KUKA KRL program: MyProgram_232().src

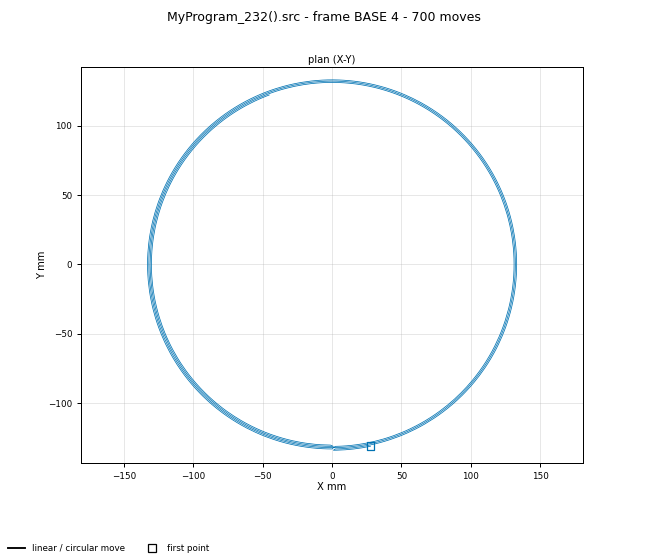
[picture p0: tool path of MyProgram_232().src in frame BASE 4, 700 of 700 moves have a stored position in this frame; points joined in program order, loops and branches not executed]
&ACCESS RVP
&REL 1
&PARAM TEMPLATE = C:\KRC\Roboter\Template\vorgabe
&PARAM EDITMASK = *
DEF MyProgram_232()
; ---- Setting reference (Base) ----
$BASE = BASE_DATA[4]

; --------------------------
; ---- Setting tool (TCP) ----
$TOOL = TOOL_DATA[3]
; --------------------------

$VEL.CP = VEL_APROX_PRINT
Startdeposition()
$VEL.CP = VEL_PRINT
LIN {X 27.6875,Y -131.1265,Z 158,A -80.2981,B 21.5066,C -0.6867,E1 21.5496,E2 528.0093} C_DIS
LIN {X 24.3865,Y -131.7813,Z 158,A -81.7242,B 21.5066,C -0.6861,E1 21.5457,E2 529.435} C_DIS
LIN {X 21.7115,Y -132.2465,Z 158,A -82.8486,B 21.5066,C -0.6869,E1 21.5426,E2 530.5558} C_DIS
LIN {X 18.7326,Y -132.701,Z 158,A -84.1707,B 21.5067,C -0.6845,E1 21.5389,E2 531.883} C_DIS
LIN {X 15.6602,Y -133.0985,Z 158,A -85.5143,B 21.5067,C -0.6828,E1 21.5352,E2 533.2299} C_DIS
LIN {X 12.3449,Y -133.4475,Z 158,A -86.8751,B 21.5067,C -0.685,E1 21.5314,E2 534.5836} C_DIS
LIN {X 9.7078,Y -133.6645,Z 158,A -88.0842,B 21.5068,C -0.681,E1 21.528,E2 535.8031} C_DIS
LIN {X 6.5931,Y -133.8544,Z 158,A -89.4325,B 21.5068,C -0.6798,E1 21.5243,E2 537.1539} C_DIS
LIN {X 3.271,Y -133.9775,Z 158,A -90.7812,B 21.5068,C -0.6827,E1 21.5205,E2 538.4945} C_DIS
LIN {X 0.9335,Y -134.0118,Z 158,A -91.4761,B 21.5063,C -0.6963,E1 21.5187,E2 539.1521} C_DIS
Enddeposition()
LIN {X 0.9335,Y -134.0118,Z 158,A -91.4761,B 21.5063,C -0.6963,E1 21.5187,E2 539.1521} C_DIS
Startdeposition()
$VEL.CP = VEL_PRINT
LIN {X 2.3152,Y -133.0672,Z 158,A -90.1607,B 20.3364,C -0.5545,E1 20.3481,E2 538.1148} C_DIS
LIN {X 6.4619,Y -132.9305,Z 158,A -88.4091,B 20.3364,C -0.5536,E1 20.353,E2 536.3665} C_DIS
LIN {X 10.2986,Y -132.6896,Z 158,A -86.7068,B 20.3364,C -0.5563,E1 20.3578,E2 534.6574} C_DIS
LIN {X 14.1975,Y -132.3277,Z 158,A -85.0987,B 20.3364,C -0.5538,E1 20.3622,E2 533.0578} C_DIS
LIN {X 17.9935,Y -131.867,Z 158,A -83.332,B 20.3363,C -0.56,E1 20.3671,E2 531.2751} C_DIS
LIN {X 21.7924,Y -131.2908,Z 158,A -81.8494,B 20.3364,C -0.5537,E1 20.3712,E2 529.8124} C_DIS
LIN {X 26.2701,Y -130.4688,Z 158,A -79.804,B 20.3364,C -0.559,E1 20.3768,E2 527.7549} C_DIS
LIN {X 29.9306,Y -129.678,Z 158,A -78.1545,B 20.3362,C -0.562,E1 20.3813,E2 526.0995} C_DIS
LIN {X 34.3931,Y -128.5662,Z 158,A -76.2181,B 20.3362,C -0.562,E1 20.3866,E2 524.1667} C_DIS
LIN {X 37.8734,Y -127.5852,Z 158,A -74.6229,B 20.3362,C -0.5654,E1 20.3908,E2 522.5654} C_DIS
LIN {X 41.9126,Y -126.315,Z 158,A -72.8787,B 20.3362,C -0.564,E1 20.3955,E2 520.8291} C_DIS
LIN {X 45.0525,Y -125.2293,Z 158,A -71.5317,B 20.3362,C -0.5621,E1 20.399,E2 519.491} C_DIS
LIN {X 48.0237,Y -124.1204,Z 158,A -70.214,B 20.3362,C -0.5618,E1 20.4024,E2 518.1778} C_DIS
LIN {X 50.4919,Y -123.1393,Z 158,A -68.8394,B 20.3359,C -0.5736,E1 20.406,E2 516.7734} C_DIS
LIN {X 54.0949,Y -121.5973,Z 158,A -67.513,B 20.3363,C -0.5601,E1 20.4093,E2 515.4899} C_DIS
LIN {X 57.1818,Y -120.1764,Z 158,A -65.8004,B 20.3359,C -0.5733,E1 20.4138,E2 513.7447} C_DIS
LIN {X 60.0472,Y -118.771,Z 158,A -64.3224,B 20.3357,C -0.5801,E1 20.4175,E2 512.2522} C_DIS
LIN {X 63.9135,Y -116.7378,Z 158,A -62.5187,B 20.3357,C -0.5798,E1 20.4219,E2 510.4559} C_DIS
LIN {X 66.8745,Y -115.0672,Z 158,A -60.0156,B 20.3343,C -0.6293,E1 20.4283,E2 507.8206} C_DIS
LIN {X 73.3086,Y -111.0787,Z 158,A -57.8118,B 20.3355,C -0.5876,E1 20.4331,E2 505.7453} C_DIS
LIN {X 76.8539,Y -108.656,Z 158,A -56.067,B 20.3355,C -0.5866,E1 20.4371,E2 504.0111} C_DIS
LIN {X 79.7409,Y -106.5556,Z 158,A -54.4115,B 20.3353,C -0.595,E1 20.4408,E2 502.3388} C_DIS
LIN {X 83.1741,Y -103.8981,Z 158,A -52.5593,B 20.3353,C -0.5982,E1 20.4449,E2 500.4862} C_DIS
LIN {X 86.5817,Y -101.0759,Z 158,A -50.6139,B 20.3351,C -0.6042,E1 20.4491,E2 498.5331} C_DIS
LIN {X 90.3656,Y -97.7078,Z 158,A -48.4774,B 20.335,C -0.6071,E1 20.4535,E2 496.3989} C_DIS
LIN {X 93.6361,Y -94.5776,Z 158,A -46.5502,B 20.3349,C -0.6107,E1 20.4573,E2 494.4717} C_DIS
LIN {X 96.0746,Y -92.0995,Z 158,A -45.0789,B 20.3349,C -0.6132,E1 20.4602,E2 493.0014} C_DIS
LIN {X 99.6884,Y -88.175,Z 158,A -42.8326,B 20.3347,C -0.6165,E1 20.4644,E2 490.7579} C_DIS
LIN {X 102.4438,Y -84.9582,Z 158,A -41.0372,B 20.3347,C -0.6199,E1 20.4676,E2 488.9632} C_DIS
LIN {X 106.2053,Y -80.2062,Z 158,A -38.3624,B 20.3343,C -0.6297,E1 20.4722,E2 486.2763} C_DIS
LIN {X 110.1173,Y -74.745,Z 158,A -35.5518,B 20.3343,C -0.6337,E1 20.4767,E2 483.4714} C_DIS
LIN {X 112.4697,Y -71.1561,Z 158,A -33.7135,B 20.3341,C -0.6384,E1 20.4795,E2 481.6312} C_DIS
LIN {X 114.6258,Y -67.6284,Z 158,A -31.9008,B 20.3339,C -0.6449,E1 20.4821,E2 479.8116} C_DIS
LIN {X 116.8267,Y -63.7505,Z 158,A -30.0164,B 20.3338,C -0.6488,E1 20.4847,E2 477.9284} C_DIS
LIN {X 118.3694,Y -60.836,Z 158,A -28.7867,B 20.3338,C -0.6442,E1 20.4862,E2 476.7201} C_DIS
LIN {X 119.8922,Y -57.7767,Z 158,A -27.2098,B 20.3336,C -0.6533,E1 20.4882,E2 475.1276} C_DIS
LIN {X 121.4292,Y -54.4706,Z 158,A -25.6532,B 20.3335,C -0.6574,E1 20.49,E2 473.5701} C_DIS
LIN {X 122.6564,Y -51.6494,Z 158,A -24.5259,B 20.3336,C -0.6523,E1 20.4912,E2 472.465} C_DIS
LIN {X 123.6856,Y -49.1368,Z 158,A -23.2765,B 20.3334,C -0.6595,E1 20.4925,E2 471.2038} C_DIS
LIN {X 124.9959,Y -45.7,Z 158,A -21.5876,B 20.3331,C -0.6691,E1 20.4942,E2 469.4993} C_DIS
LIN {X 126.2025,Y -42.2503,Z 158,A -20.0922,B 20.3331,C -0.6703,E1 20.4956,E2 468.0109} C_DIS
LIN {X 127.5193,Y -38.0983,Z 158,A -18.1166,B 20.3328,C -0.6807,E1 20.4972,E2 466.0198} C_DIS
LIN {X 128.5651,Y -34.397,Z 158,A -16.5778,B 20.3328,C -0.6805,E1 20.4983,E2 464.4928} C_DIS
LIN {X 129.3682,Y -31.2411,Z 158,A -15.2514,B 20.3328,C -0.6814,E1 20.4992,E2 463.1735} C_DIS
LIN {X 130.4065,Y -26.5763,Z 158,A -13.111,B 20.3324,C -0.6916,E1 20.5005,E2 461.0194} C_DIS
LIN {X 131.0224,Y -23.3517,Z 158,A -11.7229,B 20.3323,C -0.6949,E1 20.5012,E2 459.6321} C_DIS
LIN {X 131.6978,Y -19.1836,Z 158,A -9.8932,B 20.3321,C -0.7012,E1 20.502,E2 457.798} C_DIS
LIN {X 132.1608,Y -15.6755,Z 158,A -8.3924,B 20.332,C -0.7049,E1 20.5025,E2 456.2975} C_DIS
LIN {X 132.6069,Y -11.2968,Z 158,A -6.512,B 20.3318,C -0.7103,E1 20.503,E2 454.416} C_DIS
LIN {X 132.9005,Y -7.0583,Z 158,A -4.6718,B 20.3316,C -0.7166,E1 20.5033,E2 452.5715} C_DIS
LIN {X 133.0498,Y -3.1972,Z 158,A -2.9556,B 20.3313,C -0.7243,E1 20.5034,E2 450.8461} C_DIS
LIN {X 133.0868,Y 0.5679,Z 158,A -1.431,B 20.3313,C -0.725,E1 20.5034,E2 449.3309} C_DIS
LIN {X 133.0109,Y 4.5534,Z 158,A 0.3317,B 20.331,C -0.7325,E1 20.5034,E2 447.5598} C_DIS
LIN {X 132.8262,Y 8.3324,Z 158,A 1.8795,B 20.331,C -0.7339,E1 20.5031,E2 446.0195} C_DIS
LIN {X 132.4974,Y 12.5167,Z 158,A 3.6318,B 20.3309,C -0.7371,E1 20.5027,E2 444.2712} C_DIS
LIN {X 132.1383,Y 15.864,Z 158,A 5.101,B 20.3307,C -0.7425,E1 20.5022,E2 442.7974} C_DIS
LIN {X 131.5809,Y 19.9702,Z 158,A 6.8939,B 20.3305,C -0.7485,E1 20.5015,E2 441.0007} C_DIS
LIN {X 130.9849,Y 23.5615,Z 158,A 8.3085,B 20.3305,C -0.7463,E1 20.5008,E2 439.6028} C_DIS
LIN {X 130.4341,Y 26.4409,Z 158,A 10.0804,B 20.3296,C -0.7736,E1 20.4998,E2 437.766} C_DIS
LIN {X 129.5652,Y 30.4239,Z 158,A 11.4742,B 20.33,C -0.7623,E1 20.499,E2 436.4145} C_DIS
LIN {X 128.6379,Y 34.124,Z 158,A 13.0426,B 20.33,C -0.7639,E1 20.4979,E2 434.8528} C_DIS
LIN {X 127.7585,Y 37.2816,Z 158,A 14.6978,B 20.3294,C -0.7793,E1 20.4966,E2 433.1655} C_DIS
LIN {X 126.315,Y 41.9126,Z 158,A 16.3999,B 20.3298,C -0.7678,E1 20.4951,E2 431.5083} C_DIS
LIN {X 125.2805,Y 44.9107,Z 158,A 17.8296,B 20.3295,C -0.7748,E1 20.4938,E2 430.069} C_DIS
LIN {X 124.0786,Y 48.1311,Z 158,A 19.3211,B 20.3294,C -0.7796,E1 20.4923,E2 428.5741} C_DIS
LIN {X 122.7641,Y 51.3914,Z 158,A 20.8102,B 20.3292,C -0.7828,E1 20.4907,E2 427.0861} C_DIS
LIN {X 121.491,Y 54.3325,Z 158,A 22.195,B 20.3291,C -0.7869,E1 20.4892,E2 425.699} C_DIS
LIN {X 119.8901,Y 57.781,Z 158,A 23.9213,B 20.3288,C -0.7956,E1 20.4871,E2 423.9597} C_DIS
LIN {X 117.9529,Y 61.638,Z 158,A 25.6516,B 20.3288,C -0.7949,E1 20.4849,E2 422.243} C_DIS
LIN {X 115.9158,Y 65.3925,Z 158,A 27.571,B 20.3285,C -0.8034,E1 20.4823,E2 420.3117} C_DIS
LIN {X 113.6765,Y 69.2128,Z 158,A 29.4795,B 20.3283,C -0.8085,E1 20.4796,E2 418.4008} C_DIS
LIN {X 111.4724,Y 72.7089,Z 158,A 31.2303,B 20.3281,C -0.8118,E1 20.4769,E2 416.6517} C_DIS
LIN {X 109.0574,Y 76.2836,Z 158,A 33.094,B 20.328,C -0.8168,E1 20.474,E2 414.7853} C_DIS
LIN {X 106.4656,Y 79.8613,Z 158,A 35.0059,B 20.3278,C -0.8219,E1 20.4708,E2 412.8703} C_DIS
LIN {X 103.8172,Y 83.2749,Z 158,A 36.8027,B 20.3277,C -0.8235,E1 20.4677,E2 411.0796} C_DIS
LIN {X 101.2687,Y 86.3556,Z 158,A 38.4673,B 20.3277,C -0.8249,E1 20.4647,E2 409.4204} C_DIS
LIN {X 98.6724,Y 89.3106,Z 158,A 40.3287,B 20.3272,C -0.8362,E1 20.4612,E2 407.537} C_DIS
LIN {X 95.4044,Y 92.7938,Z 158,A 42.2848,B 20.3272,C -0.8362,E1 20.4575,E2 405.5916} C_DIS
LIN {X 92.3953,Y 95.7902,Z 158,A 44.0695,B 20.3272,C -0.8381,E1 20.4539,E2 403.8109} C_DIS
LIN {X 89.1387,Y 98.8284,Z 158,A 46.044,B 20.3269,C -0.8445,E1 20.4498,E2 401.8281} C_DIS
LIN {X 86.036,Y 101.5404,Z 158,A 47.7171,B 20.3269,C -0.8435,E1 20.4463,E2 400.1662} C_DIS
LIN {X 82.9419,Y 104.0829,Z 158,A 49.5476,B 20.3266,C -0.8514,E1 20.4423,E2 398.3217} C_DIS
LIN {X 79.1733,Y 106.9782,Z 158,A 51.5202,B 20.3266,C -0.8518,E1 20.4379,E2 396.3569} C_DIS
LIN {X 75.6862,Y 109.4731,Z 158,A 53.3873,B 20.3264,C -0.8559,E1 20.4336,E2 394.4863} C_DIS
LIN {X 71.9435,Y 111.9678,Z 158,A 55.3001,B 20.3264,C -0.8579,E1 20.4292,E2 392.5756} C_DIS
LIN {X 68.1752,Y 114.3011,Z 158,A 57.1791,B 20.3263,C -0.8595,E1 20.4247,E2 390.6993} C_DIS
LIN {X 64.1687,Y 116.5981,Z 158,A 59.1595,B 20.3262,C -0.862,E1 20.4199,E2 388.7192} C_DIS
LIN {X 60.6512,Y 118.4635,Z 158,A 60.6971,B 20.3264,C -0.8566,E1 20.4161,E2 387.2025} C_DIS
LIN {X 58.1116,Y 119.732,Z 158,A 62.1301,B 20.326,C -0.8673,E1 20.4125,E2 385.7436} C_DIS
LIN {X 54.4646,Y 121.4319,Z 158,A 63.5788,B 20.3264,C -0.8571,E1 20.4089,E2 384.3289} C_DIS
LIN {X 52.1277,Y 122.4555,Z 158,A 64.9388,B 20.3259,C -0.8696,E1 20.4053,E2 382.9371} C_DIS
LIN {X 48.5986,Y 123.8969,Z 158,A 66.4959,B 20.3259,C -0.8677,E1 20.4013,E2 381.39} C_DIS
LIN {X 45.3792,Y 125.1115,Z 158,A 67.9155,B 20.3259,C -0.8664,E1 20.3976,E2 379.9777} C_DIS
LIN {X 42.3134,Y 126.1815,Z 158,A 69.2155,B 20.3261,C -0.8634,E1 20.3942,E2 378.6895} C_DIS
LIN {X 39.1383,Y 127.202,Z 158,A 70.9018,B 20.3256,C -0.8753,E1 20.3896,E2 376.9729} C_DIS
LIN {X 35.0107,Y 128.4015,Z 158,A 72.7364,B 20.3256,C -0.8759,E1 20.3847,E2 375.1404} C_DIS
LIN {X 30.5676,Y 129.5306,Z 158,A 74.7074,B 20.3256,C -0.877,E1 20.3793,E2 373.1698} C_DIS
LIN {X 26.8773,Y 130.3453,Z 158,A 76.0752,B 20.326,C -0.8668,E1 20.3757,E2 371.8336} C_DIS
LIN {X 23.6344,Y 130.9718,Z 158,A 77.6621,B 20.3257,C -0.8745,E1 20.3713,E2 370.2271} C_DIS
LIN {X 19.8149,Y 131.6049,Z 158,A 79.2558,B 20.3257,C -0.8719,E1 20.3669,E2 368.6427} C_DIS
LIN {X 16.1677,Y 132.1021,Z 158,A 80.9086,B 20.3257,C -0.8752,E1 20.3623,E2 366.9821} C_DIS
LIN {X 12.6344,Y 132.4861,Z 158,A 82.4324,B 20.3257,C -0.8752,E1 20.3581,E2 365.4595} C_DIS
LIN {X 8.5038,Y 132.8157,Z 158,A 84.2078,B 20.3257,C -0.875,E1 20.3531,E2 363.6859} C_DIS
LIN {X 4.9454,Y 132.9956,Z 158,A 85.801,B 20.3255,C -0.8775,E1 20.3487,E2 362.0861} C_DIS
LIN {X 0.9503,Y 133.0841,Z 158,A 87.4786,B 20.3256,C -0.8755,E1 20.344,E2 360.4145} C_DIS
LIN {X -3.1981,Y 133.0498,Z 158,A 89.2834,B 20.3256,C -0.8759,E1 20.339,E2 358.6084} C_DIS
LIN {X -6.8635,Y 132.9103,Z 158,A 90.857,B 20.3256,C -0.8752,E1 20.3346,E2 357.0363} C_DIS
LIN {X -10.9849,Y 132.6333,Z 158,A 92.6045,B 20.3257,C -0.8733,E1 20.3297,E2 355.2935} C_DIS
LIN {X -15.1121,Y 132.228,Z 158,A 94.4597,B 20.3257,C -0.8753,E1 20.3246,E2 353.4312} C_DIS
LIN {X -18.8902,Y 131.7397,Z 158,A 96.0215,B 20.3257,C -0.8711,E1 20.3203,E2 351.88} C_DIS
LIN {X -21.9197,Y 131.2696,Z 158,A 97.418,B 20.3257,C -0.8734,E1 20.3164,E2 350.4751} C_DIS
LIN {X -27.1871,Y 130.2822,Z 158,A 100.1773,B 20.325,C -0.8903,E1 20.3087,E2 347.6631} C_DIS
LIN {X -31.4093,Y 129.3277,Z 158,A 101.5593,B 20.3259,C -0.8688,E1 20.3051,E2 346.3408} C_DIS
LIN {X -35.4352,Y 128.2835,Z 158,A 103.1631,B 20.3263,C -0.8595,E1 20.3008,E2 344.7609} C_DIS
LIN {X -40.955,Y 126.6295,Z 158,A 105.9418,B 20.3259,C -0.869,E1 20.2933,E2 341.9489} C_DIS
LIN {X -44.6852,Y 125.3618,Z 158,A 107.5003,B 20.3262,C -0.8613,E1 20.2893,E2 340.4086} C_DIS
LIN {X -48.125,Y 124.081,Z 158,A 109.4963,B 20.3256,C -0.8763,E1 20.2839,E2 338.3641} C_DIS
LIN {X -51.6938,Y 122.6379,Z 158,A 110.7836,B 20.3263,C -0.859,E1 20.2807,E2 337.1232} C_DIS
LIN {X -55.5799,Y 120.9258,Z 158,A 112.572,B 20.3265,C -0.8548,E1 20.2762,E2 335.3415} C_DIS
LIN {X -59.2265,Y 119.1824,Z 158,A 114.6985,B 20.3259,C -0.8678,E1 20.2708,E2 333.1705} C_DIS
LIN {X -62.4909,Y 117.5051,Z 158,A 115.9511,B 20.3266,C -0.852,E1 20.2678,E2 331.9592} C_DIS
LIN {X -66.0957,Y 115.5162,Z 158,A 117.7736,B 20.3266,C -0.851,E1 20.2633,E2 330.1328} C_DIS
LIN {X -69.6584,Y 113.4033,Z 158,A 119.5855,B 20.3266,C -0.849,E1 20.259,E2 328.3196} C_DIS
LIN {X -73.5185,Y 110.9405,Z 158,A 121.5828,B 20.3268,C -0.8464,E1 20.2543,E2 326.3217} C_DIS
LIN {X -77.0998,Y 108.4821,Z 158,A 123.4864,B 20.3268,C -0.8441,E1 20.25,E2 324.4165} C_DIS
LIN {X -80.7784,Y 105.7708,Z 158,A 125.3986,B 20.3271,C -0.838,E1 20.2457,E2 322.5136} C_DIS
LIN {X -84.0415,Y 103.1973,Z 158,A 127.2383,B 20.3271,C -0.8362,E1 20.2417,E2 320.6702} C_DIS
LIN {X -87.4428,Y 100.3313,Z 158,A 129.3036,B 20.3271,C -0.8381,E1 20.2373,E2 318.5895} C_DIS
LIN {X -91.6149,Y 96.5368,Z 158,A 131.6197,B 20.3275,C -0.8281,E1 20.2326,E2 316.2903} C_DIS
LIN {X -94.8616,Y 93.3484,Z 158,A 133.5712,B 20.3277,C -0.8232,E1 20.2287,E2 314.3425} C_DIS
LIN {X -97.9878,Y 90.061,Z 158,A 135.4847,B 20.3279,C -0.817,E1 20.2251,E2 312.4366} C_DIS
LIN {X -100.7066,Y 87.0105,Z 158,A 137.3016,B 20.328,C -0.8149,E1 20.2217,E2 310.6155} C_DIS
LIN {X -103.4772,Y 83.6965,Z 158,A 139.1697,B 20.3282,C -0.8105,E1 20.2184,E2 308.7492} C_DIS
LIN {X -106.1908,Y 80.2254,Z 158,A 141.0538,B 20.3284,C -0.8051,E1 20.2152,E2 306.8694} C_DIS
LIN {X -108.6472,Y 76.8663,Z 158,A 142.9026,B 20.3284,C -0.8026,E1 20.2122,E2 305.0166} C_DIS
LIN {X -111.157,Y 73.1897,Z 158,A 144.8114,B 20.3287,C -0.7971,E1 20.2093,E2 303.1117} C_DIS
LIN {X -113.4389,Y 69.6005,Z 158,A 146.6215,B 20.3289,C -0.7912,E1 20.2066,E2 301.307} C_DIS
LIN {X -115.6349,Y 65.8877,Z 158,A 148.4013,B 20.3292,C -0.783,E1 20.2041,E2 299.5394} C_DIS
LIN {X -117.3396,Y 62.8018,Z 158,A 150.3175,B 20.3288,C -0.7942,E1 20.2015,E2 297.5779} C_DIS
LIN {X -118.9741,Y 59.6481,Z 158,A 151.9855,B 20.3288,C -0.7953,E1 20.1994,E2 295.8955} C_DIS
LIN {X -120.7225,Y 56.0195,Z 158,A 153.2565,B 20.3296,C -0.7721,E1 20.198,E2 294.683} C_DIS
LIN {X -122.0412,Y 53.086,Z 158,A 154.4833,B 20.33,C -0.7619,E1 20.1966,E2 293.4774} C_DIS
LIN {X -123.3603,Y 49.9437,Z 158,A 156.1652,B 20.3299,C -0.7658,E1 20.1948,E2 291.7721} C_DIS
LIN {X -124.5328,Y 46.9442,Z 158,A 157.5297,B 20.33,C -0.7608,E1 20.1934,E2 290.4126} C_DIS
LIN {X -125.6883,Y 43.7559,Z 158,A 158.9927,B 20.3302,C -0.7565,E1 20.1921,E2 288.9516} C_DIS
LIN {X -126.8023,Y 40.4142,Z 158,A 160.443,B 20.3304,C -0.7493,E1 20.1908,E2 287.5116} C_DIS
LIN {X -127.5814,Y 37.8863,Z 158,A 161.7045,B 20.3304,C -0.7506,E1 20.1898,E2 286.2373} C_DIS
LIN {X -128.5518,Y 34.4471,Z 158,A 163.2055,B 20.3306,C -0.7444,E1 20.1887,E2 284.7433} C_DIS
LIN {X -129.3248,Y 31.4215,Z 158,A 165.1252,B 20.33,C -0.7627,E1 20.1874,E2 282.7565} C_DIS
LIN {X -130.3269,Y 26.9675,Z 158,A 166.484,B 20.331,C -0.7328,E1 20.1866,E2 281.4741} C_DIS
LIN {X -131.2808,Y 21.8522,Z 158,A 168.8625,B 20.331,C -0.7312,E1 20.1855,E2 279.0826} C_DIS
LIN {X -131.8295,Y 18.2618,Z 158,A 170.7093,B 20.3309,C -0.7373,E1 20.1847,E2 277.2043} C_DIS
LIN {X -132.2507,Y 14.913,Z 158,A 171.7977,B 20.3315,C -0.7185,E1 20.1844,E2 276.1622} C_DIS
LIN {X -132.6083,Y 11.28,Z 158,A 173.3574,B 20.3317,C -0.7131,E1 20.184,E2 274.6063} C_DIS
LIN {X -132.8275,Y 8.312,Z 158,A 174.7402,B 20.3317,C -0.713,E1 20.1837,E2 273.2134} C_DIS
LIN {X -133.0096,Y 4.5862,Z 158,A 176.3129,B 20.3319,C -0.7066,E1 20.1835,E2 271.6473} C_DIS
LIN {X -133.0833,Y 1.1512,Z 158,A 177.9469,B 20.3319,C -0.7079,E1 20.1835,E2 269.997} C_DIS
LIN {X -133.0505,Y -3.1741,Z 158,A 179.8024,B 20.3321,C -0.7018,E1 20.1835,E2 268.1452} C_DIS
LIN {X -132.9048,Y -6.9732,Z 158,A -178.5102,B 20.3321,C -0.6986,E1 20.1838,E2 266.4542} C_DIS
LIN {X -132.5686,Y -11.7506,Z 158,A -176.3877,B 20.3323,C -0.6945,E1 20.1842,E2 264.3274} C_DIS
LIN {X -131.6898,Y -19.2391,Z 158,A -173.2,B 20.3327,C -0.6821,E1 20.1854,E2 261.1517} C_DIS
LIN {X -131.0369,Y -23.2709,Z 158,A -170.7346,B 20.332,C -0.7045,E1 20.1866,E2 258.6029} C_DIS
LIN {X -129.9086,Y -28.9211,Z 158,A -168.8897,B 20.333,C -0.6719,E1 20.1876,E2 256.839} C_DIS
LIN {X -129.0717,Y -32.4456,Z 158,A -167.4486,B 20.3333,C -0.6626,E1 20.1886,E2 255.4144} C_DIS
LIN {X -128.21,Y -35.698,Z 158,A -165.9853,B 20.3334,C -0.6588,E1 20.1896,E2 253.9512} C_DIS
LIN {X -127.353,Y -38.6449,Z 158,A -164.6483,B 20.3335,C -0.6555,E1 20.1907,E2 252.6141} C_DIS
LIN {X -126.2959,Y -41.97,Z 158,A -163.1902,B 20.3337,C -0.6493,E1 20.192,E2 251.1634} C_DIS
LIN {X -125.0831,Y -45.4582,Z 158,A -161.2654,B 20.3335,C -0.6579,E1 20.1938,E2 249.2001} C_DIS
LIN {X -123.3883,Y -49.8743,Z 158,A -159.4866,B 20.334,C -0.6419,E1 20.1956,E2 247.4551} C_DIS
LIN {X -122.1459,Y -52.8438,Z 158,A -158.047,B 20.334,C -0.6401,E1 20.1972,E2 246.0106} C_DIS
LIN {X -120.9325,Y -55.5655,Z 158,A -156.5015,B 20.3338,C -0.6468,E1 20.199,E2 244.4349} C_DIS
LIN {X -119.5615,Y -58.4581,Z 158,A -155.4192,B 20.3343,C -0.6313,E1 20.2003,E2 243.3901} C_DIS
LIN {X -117.9903,Y -61.567,Z 158,A -153.9108,B 20.3343,C -0.6276,E1 20.2022,E2 241.8824} C_DIS
LIN {X -116.7367,Y -63.9155,Z 158,A -152.6003,B 20.3343,C -0.631,E1 20.204,E2 240.5533} C_DIS
LIN {X -114.4831,Y -67.8699,Z 158,A -150.643,B 20.3344,C -0.6257,E1 20.2067,E2 238.5985} C_DIS
LIN {X -111.8393,Y -72.1438,Z 158,A -148.3313,B 20.3344,C -0.6261,E1 20.2102,E2 236.271} C_DIS
LIN {X -108.9644,Y -76.4166,Z 158,A -146.2137,B 20.3347,C -0.6166,E1 20.2135,E2 234.1678} C_DIS
LIN {X -106.2841,Y -80.1018,Z 158,A -144.5096,B 20.3351,C -0.6015,E1 20.2163,E2 232.4969} C_DIS
LIN {X -104.1651,Y -82.8387,Z 158,A -142.7938,B 20.335,C -0.607,E1 20.2193,E2 230.755} C_DIS
LIN {X -101.4731,Y -86.1152,Z 158,A -140.8432,B 20.335,C -0.6078,E1 20.2228,E2 228.7908} C_DIS
LIN {X -98.3822,Y -89.6305,Z 158,A -138.9107,B 20.3352,C -0.6,E1 20.2264,E2 226.8701} C_DIS
LIN {X -95.3779,Y -92.8212,Z 158,A -136.9863,B 20.3352,C -0.5974,E1 20.2301,E2 224.9426} C_DIS
LIN {X -93.12,Y -95.0856,Z 158,A -135.5345,B 20.3352,C -0.5976,E1 20.233,E2 223.4826} C_DIS
LIN {X -89.6383,Y -98.3751,Z 158,A -133.5966,B 20.3355,C -0.5884,E1 20.237,E2 221.5614} C_DIS
LIN {X -86.502,Y -101.1443,Z 158,A -131.6284,B 20.3355,C -0.5917,E1 20.2412,E2 219.5739} C_DIS
LIN {X -82.7287,Y -104.2526,Z 158,A -129.6605,B 20.3357,C -0.5823,E1 20.2454,E2 217.624} C_DIS
LIN {X -79.3291,Y -106.8622,Z 158,A -127.8497,B 20.3358,C -0.5777,E1 20.2494,E2 215.8184} C_DIS
LIN {X -75.8648,Y -109.3488,Z 158,A -126.0018,B 20.3358,C -0.5751,E1 20.2536,E2 213.9699} C_DIS
LIN {X -72.3537,Y -111.703,Z 158,A -124.163,B 20.3359,C -0.573,E1 20.2579,E2 212.1297} C_DIS
LIN {X -68.9711,Y -113.8227,Z 158,A -122.3991,B 20.3359,C -0.5723,E1 20.2621,E2 210.3609} C_DIS
LIN {X -65.3056,Y -115.9646,Z 158,A -120.5566,B 20.336,C -0.5703,E1 20.2666,E2 208.5172} C_DIS
LIN {X -61.2629,Y -118.1499,Z 158,A -118.5404,B 20.336,C -0.5693,E1 20.2716,E2 206.4969} C_DIS
LIN {X -57.7364,Y -119.9114,Z 158,A -116.938,B 20.3362,C -0.5633,E1 20.2756,E2 204.9064} C_DIS
LIN {X -55.1469,Y -121.126,Z 158,A -115.7385,B 20.3362,C -0.5606,E1 20.2786,E2 203.7113} C_DIS
LIN {X -51.7049,Y -122.6332,Z 158,A -114.0563,B 20.3362,C -0.5615,E1 20.2829,E2 202.0213} C_DIS
LIN {X -48.3353,Y -123.9993,Z 158,A -112.5527,B 20.3363,C -0.5574,E1 20.2868,E2 200.5254} C_DIS
LIN {X -45.159,Y -125.1909,Z 158,A -111.2595,B 20.3366,C -0.5491,E1 20.2902,E2 199.2529} C_DIS
LIN {X -42.247,Y -126.2036,Z 158,A -109.5341,B 20.3362,C -0.5647,E1 20.2949,E2 197.4785} C_DIS
LIN {X -37.7094,Y -127.6332,Z 158,A -107.6664,B 20.3364,C -0.5556,E1 20.2998,E2 195.6331} C_DIS
LIN {X -33.5852,Y -128.7813,Z 158,A -105.7864,B 20.3364,C -0.5559,E1 20.3049,E2 193.7485} C_DIS
LIN {X -30.1706,Y -129.6232,Z 158,A -104.2068,B 20.3364,C -0.5579,E1 20.3092,E2 192.1606} C_DIS
LIN {X -26.2591,Y -130.4711,Z 158,A -102.5329,B 20.3364,C -0.555,E1 20.3137,E2 190.4925} C_DIS
LIN {X -22.3213,Y -131.2026,Z 158,A -100.8676,B 20.3364,C -0.5519,E1 20.3183,E2 188.8341} C_DIS
LIN {X -18.9064,Y -131.7374,Z 158,A -99.4015,B 20.3365,C -0.5506,E1 20.3223,E2 187.3702} C_DIS
LIN {X -15.1281,Y -132.2261,Z 158,A -97.6353,B 20.3364,C -0.5556,E1 20.3273,E2 185.5881} C_DIS
LIN {X -11.2945,Y -132.6071,Z 158,A -96.0487,B 20.3364,C -0.5524,E1 20.3317,E2 184.0097} C_DIS
LIN {X -7.1827,Y -132.8942,Z 158,A -94.2753,B 20.3364,C -0.5524,E1 20.3366,E2 182.2357} C_DIS
LIN {X -3.5627,Y -133.0397,Z 158,A -92.7354,B 20.3365,C -0.5516,E1 20.3409,E2 180.6975} C_DIS
LIN {X -0.0281,Y -133.0892,Z 158,A -91.0677,B 20.3363,C -0.5582,E1 20.3456,E2 179.0111} C_DIS
LIN {X -0.0281,Y -133.0892,Z 158,A -91.0677,B 20.3363,C -0.5582,E1 20.3456,E2 179.0111} C_DIS
Enddeposition()
LIN {X 0.9243,Y -132.1538,Z 158,A -91.1186,B 19.1216,C -0.3755,E1 19.1257,E2 179.4916} C_DIS
Startdeposition()
$VEL.CP = VEL_PRINT
LIN {X -3.0717,Y -132.1236,Z 158,A -92.9298,B 19.1216,C -0.3722,E1 19.1206,E2 181.3132} C_DIS
LIN {X -6.9071,Y -131.9776,Z 158,A -94.5438,B 19.1216,C -0.3741,E1 19.1161,E2 182.9218} C_DIS
LIN {X -11.0301,Y -131.6968,Z 158,A -96.3303,B 19.1216,C -0.3744,E1 19.1111,E2 184.7083} C_DIS
LIN {X -15.0739,Y -131.2967,Z 158,A -98.189,B 19.1216,C -0.3708,E1 19.1059,E2 186.5794} C_DIS
LIN {X -19.1415,Y -130.765,Z 158,A -99.9299,B 19.1216,C -0.3727,E1 19.1011,E2 188.3163} C_DIS
LIN {X -22.1969,Y -130.2811,Z 158,A -101.2675,B 19.1216,C -0.3733,E1 19.0975,E2 189.6538} C_DIS
LIN {X -26.1878,Y -129.5372,Z 158,A -103.0403,B 19.1216,C -0.3735,E1 19.0926,E2 191.4284} C_DIS
LIN {X -30.1532,Y -128.6739,Z 158,A -104.818,B 19.1216,C -0.3737,E1 19.0877,E2 193.2087} C_DIS
LIN {X -36.3455,Y -127.0639,Z 158,A -108.2022,B 19.122,C -0.3521,E1 19.0784,E2 196.6659} C_DIS
LIN {X -41.3929,Y -125.5085,Z 158,A -109.6946,B 19.1214,C -0.3844,E1 19.0747,E2 198.0631} C_DIS
LIN {X -44.7029,Y -124.3675,Z 158,A -111.3487,B 19.1214,C -0.3805,E1 19.0703,E2 199.7336} C_DIS
LIN {X -48.2277,Y -123.044,Z 158,A -112.9646,B 19.1214,C -0.3827,E1 19.0661,E2 201.3474} C_DIS
LIN {X -52.4931,Y -121.2851,Z 158,A -114.953,B 19.1214,C -0.3852,E1 19.061,E2 203.3341} C_DIS
LIN {X -55.6734,Y -119.8587,Z 158,A -116.4353,B 19.1214,C -0.388,E1 19.0572,E2 204.8127} C_DIS
LIN {X -58.4844,Y -118.5122,Z 158,A -117.8215,B 19.1214,C -0.3883,E1 19.0537,E2 206.2028} C_DIS
LIN {X -61.4044,Y -117.026,Z 158,A -119.2698,B 19.1214,C -0.3891,E1 19.0501,E2 207.6541} C_DIS
LIN {X -64.8462,Y -115.1568,Z 158,A -121.0525,B 19.1214,C -0.3881,E1 19.0458,E2 209.4465} C_DIS
LIN {X -69.37,Y -112.49,Z 158,A -123.2546,B 19.1212,C -0.3942,E1 19.0405,E2 211.6389} C_DIS
LIN {X -72.8252,Y -110.2843,Z 158,A -125.1126,B 19.1212,C -0.394,E1 19.0361,E2 213.5058} C_DIS
LIN {X -76.5425,Y -107.7381,Z 158,A -127.0467,B 19.1212,C -0.3979,E1 19.0317,E2 215.4368} C_DIS
LIN {X -79.6588,Y -105.4542,Z 158,A -128.7385,B 19.1211,C -0.4001,E1 19.0279,E2 217.1298} C_DIS
LIN {X -83.0254,Y -102.8246,Z 158,A -131.2243,B 19.1215,C -0.3801,E1 19.0224,E2 219.6896} C_DIS
LIN {X -87.0758,Y -99.4181,Z 158,A -132.6948,B 19.1208,C -0.4148,E1 19.0195,E2 221.0611} C_DIS
LIN {X -89.3353,Y -97.3926,Z 158,A -134.7295,B 19.1213,C -0.3909,E1 19.0151,E2 223.1804} C_DIS
LIN {X -92.709,Y -94.187,Z 158,A -136.0353,B 19.1207,C -0.4212,E1 19.0127,E2 224.4004} C_DIS
LIN {X -95.0384,Y -91.8358,Z 158,A -137.7163,B 19.1207,C -0.4151,E1 19.0093,E2 226.1098} C_DIS
LIN {X -98.1207,Y -88.5356,Z 158,A -140.1686,B 19.1211,C -0.4013,E1 19.0046,E2 228.619} C_DIS
LIN {X -101.1465,Y -85.0618,Z 158,A -141.5192,B 19.1205,C -0.4295,E1 19.0023,E2 229.8915} C_DIS
LIN {X -104.636,Y -80.731,Z 158,A -144.0341,B 19.1205,C -0.4313,E1 18.9979,E2 232.4168} C_DIS
LIN {X -106.8888,Y -77.7234,Z 158,A -145.6676,B 19.1204,C -0.435,E1 18.9952,E2 234.0493} C_DIS
LIN {X -109.206,Y -74.4334,Z 158,A -148.0698,B 19.1208,C -0.4155,E1 18.9913,E2 236.5274} C_DIS
LIN {X -111.9227,Y -70.2816,Z 158,A -149.4872,B 19.1201,C -0.4475,E1 18.9893,E2 237.8562} C_DIS
LIN {X -113.7355,Y -67.309,Z 158,A -151.5622,B 19.1204,C -0.431,E1 18.9862,E2 239.9965} C_DIS
LIN {X -115.6955,Y -63.8803,Z 158,A -152.6905,B 19.1199,C -0.4566,E1 18.9848,E2 241.054} C_DIS
LIN {X -117.1115,Y -61.2415,Z 158,A -154.1487,B 19.1199,C -0.4543,E1 18.9828,E2 242.5297} C_DIS
LIN {X -118.5614,Y -58.3847,Z 158,A -156.425,B 19.1205,C -0.4263,E1 18.9799,E2 244.9087} C_DIS
LIN {X -121.1721,Y -52.7543,Z 158,A -158.0577,B 19.1195,C -0.4716,E1 18.9782,E2 246.414} C_DIS
LIN {X -122.3099,Y -50.0638,Z 158,A -160.2817,B 19.1202,C -0.4409,E1 18.9757,E2 248.7493} C_DIS
LIN {X -124.2631,Y -44.9925,Z 158,A -161.6482,B 19.1192,C -0.483,E1 18.9745,E2 249.9965} C_DIS
LIN {X -125.5043,Y -41.4056,Z 158,A -163.6661,B 19.1195,C -0.4744,E1 18.9726,E2 252.0564} C_DIS
LIN {X -126.8102,Y -37.2131,Z 158,A -165.4728,B 19.1192,C -0.4834,E1 18.9712,E2 253.8493} C_DIS
LIN {X -127.6752,Y -34.1276,Z 158,A -166.8673,B 19.1192,C -0.4874,E1 18.9701,E2 255.2426} C_DIS
LIN {X -128.4759,Y -30.9772,Z 158,A -168.3591,B 19.1192,C -0.4886,E1 18.9691,E2 256.7423} C_DIS
LIN {X -129.8258,Y -24.7167,Z 158,A -171.3032,B 19.119,C -0.4911,E1 18.9675,E2 259.7023} C_DIS
LIN {X -130.5172,Y -20.7665,Z 158,A -173.1436,B 19.119,C -0.4927,E1 18.9666,E2 261.5523} C_DIS
LIN {X -131.3961,Y -14.1695,Z 158,A -175.646,B 19.1184,C -0.5152,E1 18.9658,E2 264.0056} C_DIS
LIN {X -131.8925,Y -8.3762,Z 158,A -178.3422,B 19.1184,C -0.5168,E1 18.9652,E2 266.719} C_DIS
LIN {X -132.0793,Y -4.5924,Z 158,A -179.9322,B 19.1182,C -0.5237,E1 18.965,E2 268.3004} C_DIS
LIN {X -132.1578,Y 0.521,Z 158,A 177.3791,B 19.1185,C -0.514,E1 18.965,E2 271.041} C_DIS
LIN {X -132.0863,Y 4.4127,Z 158,A 176.0068,B 19.118,C -0.5303,E1 18.965,E2 272.374} C_DIS
LIN {X -131.8989,Y 8.2723,Z 158,A 174.3801,B 19.1179,C -0.5373,E1 18.9653,E2 273.9924} C_DIS
LIN {X -131.5037,Y 13.1431,Z 158,A 172.215,B 19.1177,C -0.5423,E1 18.9658,E2 276.1598} C_DIS
LIN {X -130.9973,Y 17.4784,Z 158,A 170.3488,B 19.1175,C -0.5491,E1 18.9665,E2 278.0201} C_DIS
LIN {X -129.7536,Y 25.0947,Z 158,A 167.0822,B 19.1172,C -0.5623,E1 18.968,E2 281.2722} C_DIS
LIN {X -128.909,Y 29.124,Z 158,A 165.061,B 19.1172,C -0.5594,E1 18.9692,E2 283.3184} C_DIS
LIN {X -127.8041,Y 33.644,Z 158,A 163.0312,B 19.1171,C -0.5651,E1 18.9706,E2 285.3466} C_DIS
LIN {X -126.771,Y 37.3468,Z 158,A 161.4792,B 19.1168,C -0.5742,E1 18.9718,E2 286.8826} C_DIS
LIN {X -125.7783,Y 40.5657,Z 158,A 160.0557,B 19.1167,C -0.58,E1 18.9729,E2 288.2994} C_DIS
LIN {X -124.7982,Y 43.4863,Z 158,A 158.6746,B 19.1166,C -0.5824,E1 18.9742,E2 289.6838} C_DIS
LIN {X -123.5001,Y 47.0521,Z 158,A 156.8306,B 19.1166,C -0.5802,E1 18.976,E2 291.5485} C_DIS
LIN {X -121.9094,Y 51.0266,Z 158,A 155.0689,B 19.1164,C -0.589,E1 18.9779,E2 293.2963} C_DIS
LIN {X -120.4527,Y 54.3779,Z 158,A 153.5193,B 19.1162,C -0.5948,E1 18.9796,E2 294.8394} C_DIS
LIN {X -118.7841,Y 57.9318,Z 158,A 151.7988,B 19.1161,C -0.5991,E1 18.9817,E2 296.5594} C_DIS
LIN {X -117.3104,Y 60.8628,Z 158,A 149.9259,B 19.1164,C -0.5871,E1 18.9841,E2 298.4826} C_DIS
LIN {X -115.3991,Y 64.4151,Z 158,A 148.4868,B 19.116,C -0.603,E1 18.986,E2 299.8831} C_DIS
LIN {X -113.2266,Y 68.161,Z 158,A 146.639,B 19.1158,C -0.6092,E1 18.9886,E2 301.7246} C_DIS
LIN {X -111.0252,Y 71.6911,Z 158,A 144.7787,B 19.1157,C -0.6121,E1 18.9914,E2 303.5888} C_DIS
LIN {X -108.6018,Y 75.3114,Z 158,A 142.9223,B 19.1155,C -0.6183,E1 18.9943,E2 305.4386} C_DIS
LIN {X -106.1754,Y 78.6955,Z 158,A 141.0961,B 19.1154,C -0.6222,E1 18.9973,E2 307.2645} C_DIS
LIN {X -103.7453,Y 81.8725,Z 158,A 139.3663,B 19.1152,C -0.6268,E1 19.0003,E2 308.9913} C_DIS
LIN {X -101.2272,Y 84.9656,Z 158,A 137.6063,B 19.1152,C -0.63,E1 19.0034,E2 310.7524} C_DIS
LIN {X -98.2258,Y 88.4189,Z 158,A 135.602,B 19.115,C -0.6341,E1 19.0071,E2 312.7562} C_DIS
LIN {X -95.2654,Y 91.6011,Z 158,A 133.7284,B 19.1148,C -0.6389,E1 19.0107,E2 314.626} C_DIS
LIN {X -92.331,Y 94.5577,Z 158,A 131.5843,B 19.1151,C -0.6309,E1 19.0151,E2 316.8069} C_DIS
LIN {X -89.649,Y 97.1038,Z 158,A 130.5198,B 19.1144,C -0.6539,E1 19.0171,E2 317.8064} C_DIS
LIN {X -87.7334,Y 98.8384,Z 158,A 129.151,B 19.1146,C -0.6474,E1 19.02,E2 319.2028} C_DIS
LIN {X -84.4737,Y 101.6383,Z 158,A 127.2594,B 19.1145,C -0.6503,E1 19.024,E2 321.0953} C_DIS
LIN {X -81.0049,Y 104.4237,Z 158,A 125.3352,B 19.1143,C -0.6544,E1 19.0282,E2 323.0165} C_DIS
LIN {X -77.4687,Y 107.0734,Z 158,A 123.4759,B 19.1141,C -0.6602,E1 19.0324,E2 324.8667} C_DIS
LIN {X -74.3832,Y 109.24,Z 158,A 121.7221,B 19.1141,C -0.6589,E1 19.0365,E2 326.6324} C_DIS
LIN {X -70.7694,Y 111.6148,Z 158,A 119.8687,B 19.1141,C -0.6631,E1 19.0408,E2 328.4811} C_DIS
LIN {X -66.9991,Y 113.9177,Z 158,A 117.9343,B 19.114,C -0.6657,E1 19.0454,E2 330.4153} C_DIS
LIN {X -63.0211,Y 116.166,Z 158,A 115.0146,B 19.115,C -0.6346,E1 19.0529,E2 333.4414} C_DIS
LIN {X -56.8118,Y 119.3232,Z 158,A 113.3283,B 19.1132,C -0.6882,E1 19.0567,E2 334.9696} C_DIS
LIN {X -48.656,Y 122.8774,Z 158,A 109.169,B 19.1134,C -0.682,E1 19.0675,E2 339.1608} C_DIS
LIN {X -44.6931,Y 124.371,Z 158,A 107.2772,B 19.1134,C -0.6822,E1 19.0724,E2 341.0573} C_DIS
LIN {X -41.6057,Y 125.4377,Z 158,A 105.2439,B 19.1141,C -0.6608,E1 19.078,E2 343.161} C_DIS
LIN {X -36.7879,Y 126.9347,Z 158,A 103.6961,B 19.1132,C -0.6869,E1 19.0819,E2 344.6326} C_DIS
LIN {X -32.6746,Y 128.0548,Z 158,A 101.0949,B 19.1141,C -0.6604,E1 19.0892,E2 347.3198} C_DIS
LIN {X -27.1808,Y 129.3344,Z 158,A 99.4184,B 19.1131,C -0.6912,E1 19.0935,E2 348.905} C_DIS
LIN {X -21.3147,Y 130.4284,Z 158,A 96.858,B 19.113,C -0.694,E1 19.1005,E2 351.4604} C_DIS
LIN {X -18.3142,Y 130.8832,Z 158,A 95.3619,B 19.1132,C -0.6879,E1 19.1047,E2 352.9767} C_DIS
LIN {X -12.8043,Y 131.5362,Z 158,A 93.054,B 19.113,C -0.6928,E1 19.1111,E2 355.2716} C_DIS
LIN {X -9.3058,Y 131.8302,Z 158,A 91.5468,B 19.113,C -0.6939,E1 19.1153,E2 356.7762} C_DIS
LIN {X -5.2365,Y 132.0542,Z 158,A 89.7729,B 19.113,C -0.6941,E1 19.1202,E2 358.5499} C_DIS
LIN {X -1.262,Y 132.1531,Z 158,A 87.9771,B 19.113,C -0.6917,E1 19.1253,E2 360.3533} C_DIS
LIN {X 2.8395,Y 132.129,Z 158,A 86.2304,B 19.113,C -0.6931,E1 19.1301,E2 362.0955} C_DIS
LIN {X 6.5933,Y 131.9934,Z 158,A 84.6453,B 19.113,C -0.6948,E1 19.1345,E2 363.6748} C_DIS
LIN {X 10.3491,Y 131.7541,Z 158,A 82.8687,B 19.1132,C -0.689,E1 19.1395,E2 365.4679} C_DIS
LIN {X 14.29,Y 131.3831,Z 158,A 81.2893,B 19.113,C -0.694,E1 19.1439,E2 367.0305} C_DIS
LIN {X 19.4332,Y 130.7233,Z 158,A 78.9202,B 19.1132,C -0.6886,E1 19.1505,E2 369.4133} C_DIS
LIN {X 23.3271,Y 130.0827,Z 158,A 77.3583,B 19.113,C -0.6938,E1 19.1547,E2 370.9572} C_DIS
LIN {X 26.6668,Y 129.4397,Z 158,A 75.7716,B 19.1132,C -0.6887,E1 19.1591,E2 372.5569} C_DIS
LIN {X 32.9645,Y 127.9813,Z 158,A 73.2589,B 19.1128,C -0.6984,E1 19.1658,E2 375.035} C_DIS
LIN {X 38.3626,Y 126.4676,Z 158,A 70.5753,B 19.1132,C -0.6867,E1 19.1731,E2 377.7484} C_DIS
LIN {X 41.9849,Y 125.3114,Z 158,A 69.0251,B 19.1132,C -0.6892,E1 19.1772,E2 379.287} C_DIS
LIN {X 44.9277,Y 124.2865,Z 158,A 67.6332,B 19.1132,C -0.6863,E1 19.1809,E2 380.6838} C_DIS
LIN {X 48.4668,Y 122.951,Z 158,A 66.0648,B 19.1132,C -0.6875,E1 19.1849,E2 382.2439} C_DIS
LIN {X 51.0348,Y 121.9059,Z 158,A 64.8011,B 19.1133,C -0.6838,E1 19.1882,E2 383.515} C_DIS
LIN {X 54.1015,Y 120.5763,Z 158,A 63.4031,B 19.1133,C -0.6842,E1 19.1918,E2 384.9072} C_DIS
LIN {X 57.1331,Y 119.1698,Z 158,A 61.9395,B 19.1134,C -0.6819,E1 19.1955,E2 386.3728} C_DIS
LIN {X 60.742,Y 117.3738,Z 158,A 60.1143,B 19.1136,C -0.6765,E1 19.2,E2 388.2077} C_DIS
LIN {X 64.4091,Y 115.4025,Z 158,A 58.3831,B 19.1136,C -0.677,E1 19.2043,E2 389.9306} C_DIS
LIN {X 67.9767,Y 113.3376,Z 158,A 56.5133,B 19.1138,C -0.671,E1 19.2088,E2 391.8109} C_DIS
LIN {X 71.6751,Y 111.0356,Z 158,A 54.6502,B 19.1138,C -0.6691,E1 19.2132,E2 393.6716} C_DIS
LIN {X 75.227,Y 108.6604,Z 158,A 52.8943,B 19.1138,C -0.67,E1 19.2172,E2 395.4169} C_DIS
LIN {X 78.5167,Y 106.3078,Z 158,A 51.0836,B 19.114,C -0.6647,E1 19.2213,E2 397.2352} C_DIS
LIN {X 83.4488,Y 102.4815,Z 158,A 48.6154,B 19.1138,C -0.6694,E1 19.2267,E2 399.6766} C_DIS
LIN {X 85.8808,Y 100.4526,Z 158,A 47.0345,B 19.1142,C -0.6583,E1 19.2301,E2 401.283} C_DIS
LIN {X 88.8208,Y 97.862,Z 158,A 45.5384,B 19.114,C -0.6633,E1 19.2332,E2 402.7561} C_DIS
LIN {X 91.0615,Y 95.7811,Z 158,A 43.9447,B 19.1145,C -0.6496,E1 19.2365,E2 404.3825} C_DIS
LIN {X 94.1625,Y 92.734,Z 158,A 42.0908,B 19.1145,C -0.6469,E1 19.2402,E2 406.2341} C_DIS
LIN {X 98.2535,Y 88.388,Z 158,A 39.5851,B 19.1147,C -0.6446,E1 19.2449,E2 408.732} C_DIS
LIN {X 100.9929,Y 85.2449,Z 158,A 37.7019,B 19.1149,C -0.6374,E1 19.2483,E2 410.6256} C_DIS
LIN {X 103.5432,Y 82.1277,Z 158,A 35.9898,B 19.1149,C -0.6347,E1 19.2513,E2 412.3351} C_DIS
LIN {X 106.2799,Y 78.5547,Z 158,A 34.1179,B 19.115,C -0.6333,E1 19.2545,E2 414.1993} C_DIS
LIN {X 108.3879,Y 75.6188,Z 158,A 32.623,B 19.115,C -0.6324,E1 19.2569,E2 415.6871} C_DIS
LIN {X 110.5804,Y 72.3754,Z 158,A 30.8616,B 19.1153,C -0.6255,E1 19.2596,E2 417.4578} C_DIS
LIN {X 112.8625,Y 68.7628,Z 158,A 28.9978,B 19.1154,C -0.6202,E1 19.2624,E2 419.3248} C_DIS
LIN {X 115.0463,Y 65.0428,Z 158,A 27.1227,B 19.1156,C -0.6151,E1 19.265,E2 421.2025} C_DIS
LIN {X 117.1203,Y 61.2247,Z 158,A 25.3263,B 19.1156,C -0.6137,E1 19.2673,E2 422.9903} C_DIS
LIN {X 118.667,Y 58.1708,Z 158,A 23.8943,B 19.1156,C -0.6118,E1 19.2691,E2 424.4177} C_DIS
LIN {X 120.1216,Y 55.1048,Z 158,A 22.4619,B 19.1158,C -0.6094,E1 19.2708,E2 425.8471} C_DIS
LIN {X 121.3697,Y 52.2975,Z 158,A 21.0897,B 19.1159,C -0.604,E1 19.2723,E2 427.2257} C_DIS
LIN {X 122.7208,Y 49.0446,Z 158,A 19.4892,B 19.1162,C -0.5966,E1 19.274,E2 428.8368} C_DIS
LIN {X 124.3382,Y 44.7842,Z 158,A 17.6168,B 19.1162,C -0.5952,E1 19.2758,E2 430.6993} C_DIS
LIN {X 125.5816,Y 41.1735,Z 158,A 16.0059,B 19.1162,C -0.5923,E1 19.2773,E2 432.3069} C_DIS
LIN {X 127.1433,Y 36.0617,Z 158,A 13.8206,B 19.1163,C -0.591,E1 19.279,E2 434.4793} C_DIS
LIN {X 127.74,Y 33.8846,Z 158,A 11.7374,B 19.1177,C -0.5418,E1 19.2806,E2 436.6955} C_DIS
LIN {X 129.3192,Y 27.2514,Z 158,A 9.4465,B 19.1172,C -0.5606,E1 19.2819,E2 438.9115} C_DIS
LIN {X 129.9804,Y 23.8989,Z 158,A 8.3938,B 19.1168,C -0.5742,E1 19.2824,E2 439.9147} C_DIS
LIN {X 130.6631,Y 19.8243,Z 158,A 6.4555,B 19.1172,C -0.5625,E1 19.2833,E2 441.8732} C_DIS
LIN {X 131.1835,Y 16.0227,Z 158,A 4.8317,B 19.1172,C -0.559,E1 19.2839,E2 443.4946} C_DIS
LIN {X 131.5993,Y 12.1476,Z 158,A 3.0885,B 19.1175,C -0.5515,E1 19.2844,E2 445.2466} C_DIS
LIN {X 131.9121,Y 8.0573,Z 158,A 1.4408,B 19.1175,C -0.5515,E1 19.2847,E2 446.8812} C_DIS
LIN {X 132.0991,Y 3.9536,Z 158,A -0.4038,B 19.1177,C -0.5433,E1 19.2849,E2 448.736} C_DIS
LIN {X 132.1587,Y -0.3527,Z 158,A -2.2468,B 19.1178,C -0.5385,E1 19.2849,E2 450.579} C_DIS
LIN {X 132.0897,Y -4.2917,Z 158,A -3.9849,B 19.118,C -0.5319,E1 19.2848,E2 452.3233} C_DIS
LIN {X 131.8804,Y -8.5723,Z 158,A -5.8345,B 19.1181,C -0.5264,E1 19.2845,E2 454.1747} C_DIS
LIN {X 131.3455,Y -14.6389,Z 158,A -8.1877,B 19.1181,C -0.5304,E1 19.2839,E2 456.4972} C_DIS
LIN {X 130.8229,Y -18.7364,Z 158,A -10.1163,B 19.1183,C -0.5189,E1 19.2832,E2 458.4452} C_DIS
LIN {X 129.9853,Y -23.8714,Z 158,A -12.4417,B 19.1186,C -0.5089,E1 19.2821,E2 460.7826} C_DIS
LIN {X 128.5074,Y -30.8466,Z 158,A -15.3995,B 19.1186,C -0.505,E1 19.2803,E2 463.7291} C_DIS
LIN {X 127.6389,Y -34.2638,Z 158,A -17.641,B 19.1196,C -0.4702,E1 19.2786,E2 466.0587} C_DIS
LIN {X 126.0999,Y -39.5588,Z 158,A -19.2322,B 19.1189,C -0.4967,E1 19.2774,E2 467.5576} C_DIS
LIN {X 125.2093,Y -42.2916,Z 158,A -20.4877,B 19.119,C -0.4925,E1 19.2763,E2 468.8161} C_DIS
LIN {X 124.1997,Y -45.1684,Z 158,A -22.552,B 19.1199,C -0.4572,E1 19.2742,E2 470.9719} C_DIS
LIN {X 122.2257,Y -50.2691,Z 158,A -24.1418,B 19.1192,C -0.4831,E1 19.2727,E2 472.4714} C_DIS
LIN {X 120.5219,Y -54.223,Z 158,A -26.0312,B 19.1194,C -0.4767,E1 19.2706,E2 474.3664} C_DIS
LIN {X 119.002,Y -57.4842,Z 158,A -27.7885,B 19.1197,C -0.4638,E1 19.2684,E2 476.1501} C_DIS
LIN {X 117.1957,Y -61.0811,Z 158,A -29.3199,B 19.1197,C -0.4679,E1 19.2665,E2 477.6583} C_DIS
LIN {X 115.341,Y -64.5185,Z 158,A -31.0888,B 19.1197,C -0.4599,E1 19.2641,E2 479.439} C_DIS
LIN {X 113.1935,Y -68.2157,Z 158,A -32.9205,B 19.1199,C -0.4556,E1 19.2615,E2 481.2709} C_DIS
LIN {X 110.9869,Y -71.7501,Z 158,A -34.6588,B 19.1199,C -0.4536,E1 19.2589,E2 483.0037} C_DIS
LIN {X 108.9661,Y -74.7829,Z 158,A -36.7419,B 19.1205,C -0.4282,E1 19.2555,E2 485.1499} C_DIS
LIN {X 106.3569,Y -78.4497,Z 158,A -38.9403,B 19.1208,C -0.4128,E1 19.2518,E2 487.3809} C_DIS
LIN {X 102.7865,Y -83.0726,Z 158,A -40.6305,B 19.1202,C -0.4415,E1 19.2491,E2 488.9734} C_DIS
LIN {X 97.5416,Y -89.1732,Z 158,A -44.6623,B 19.1209,C -0.4101,E1 19.2415,E2 493.076} C_DIS
LIN {X 94.4619,Y -92.4288,Z 158,A -46.0136,B 19.1205,C -0.4302,E1 19.239,E2 494.3586} C_DIS
LIN {X 91.7164,Y -95.154,Z 158,A -48.2394,B 19.121,C -0.4035,E1 19.2344,E2 496.653} C_DIS
LIN {X 88.4831,Y -98.1683,Z 158,A -50.2682,B 19.1212,C -0.3946,E1 19.2302,E2 498.6979} C_DIS
LIN {X 84.6807,Y -101.4663,Z 158,A -51.8006,B 19.1207,C -0.4168,E1 19.2271,E2 500.155} C_DIS
LIN {X 81.6717,Y -103.9031,Z 158,A -53.6433,B 19.121,C -0.4064,E1 19.223,E2 502.0197} C_DIS
LIN {X 76.4472,Y -107.8055,Z 158,A -56.3809,B 19.121,C -0.4045,E1 19.2168,E2 504.7501} C_DIS
LIN {X 72.8831,Y -110.2462,Z 158,A -58.5919,B 19.1213,C -0.387,E1 19.2116,E2 507.0042} C_DIS
LIN {X 69.4759,Y -112.4243,Z 158,A -60.0833,B 19.1212,C -0.3946,E1 19.2081,E2 508.4663} C_DIS
LIN {X 66.3038,Y -114.3237,Z 158,A -61.554,B 19.1212,C -0.3973,E1 19.2046,E2 509.9228} C_DIS
LIN {X 62.6065,Y -116.3896,Z 158,A -63.9492,B 19.1216,C -0.3714,E1 19.1986,E2 512.3874} C_DIS
LIN {X 58.2074,Y -118.6489,Z 158,A -65.4628,B 19.1212,C -0.3938,E1 19.195,E2 513.8275} C_DIS
LIN {X 55.2834,Y -120.039,Z 158,A -66.8632,B 19.1212,C -0.3918,E1 19.1914,E2 515.229} C_DIS
LIN {X 51.3612,Y -121.7696,Z 158,A -68.7584,B 19.1213,C -0.3877,E1 19.1865,E2 517.1307} C_DIS
LIN {X 48.0343,Y -123.1192,Z 158,A -70.3227,B 19.1213,C -0.3853,E1 19.1825,E2 518.6974} C_DIS
LIN {X 43.8904,Y -124.6582,Z 158,A -72.2518,B 19.1214,C -0.3824,E1 19.1774,E2 520.6299} C_DIS
LIN {X 38.3754,Y -126.4636,Z 158,A -74.8146,B 19.1215,C -0.3777,E1 19.1706,E2 523.2007} C_DIS
LIN {X 33.8521,Y -127.7487,Z 158,A -76.6675,B 19.1215,C -0.3831,E1 19.1656,E2 525.033} C_DIS
LIN {X 30.472,Y -128.5977,Z 158,A -78.3295,B 19.1215,C -0.3757,E1 19.1611,E2 526.7144} C_DIS
LIN {X 24.1189,Y -129.9402,Z 158,A -81.0377,B 19.1215,C -0.3777,E1 19.1537,E2 529.412} C_DIS
LIN {X 20.9935,Y -130.4819,Z 158,A -82.5269,B 19.1216,C -0.3721,E1 19.1495,E2 530.916} C_DIS
LIN {X 17.0598,Y -131.0521,Z 158,A -84.1099,B 19.1216,C -0.3767,E1 19.1452,E2 532.4832} C_DIS
LIN {X 13.1134,Y -131.5066,Z 158,A -85.8876,B 19.1216,C -0.3736,E1 19.1403,E2 534.2687} C_DIS
LIN {X 9.2051,Y -131.8376,Z 158,A -87.6143,B 19.1216,C -0.3718,E1 19.1354,E2 535.9997} C_DIS
LIN {X 5.3759,Y -132.0488,Z 158,A -89.2569,B 19.1216,C -0.3721,E1 19.1309,E2 537.6408} C_DIS
LIN {X 0.9243,Y -132.1538,Z 158,A -91.1155,B 19.1216,C -0.3745,E1 19.1257,E2 539.4916} C_DIS
Enddeposition()
LIN {X 0.9243,Y -132.1538,Z 158,A -91.1155,B 19.1216,C -0.3745,E1 19.1257,E2 539.4916} C_DIS
Startdeposition()
$VEL.CP = VEL_PRINT
LIN {X 2.341,Y -131.2079,Z 158,A -89.3177,B 17.734,C -0.2522,E1 17.7405,E2 537.9706} C_DIS
LIN {X 6.4236,Y -131.0714,Z 158,A -87.6219,B 17.734,C -0.2494,E1 17.7452,E2 536.2845} C_DIS
LIN {X 10.2993,Y -130.8259,Z 158,A -85.8318,B 17.734,C -0.2536,E1 17.7502,E2 534.482} C_DIS
LIN {X 14.1697,Y -130.4614,Z 158,A -84.2119,B 17.734,C -0.2516,E1 17.7547,E2 532.8703} C_DIS
LIN {X 18.3546,Y -129.9387,Z 158,A -82.4466,B 17.734,C -0.2498,E1 17.7595,E2 531.113} C_DIS
LIN {X 21.4734,Y -129.4597,Z 158,A -81.1419,B 17.734,C -0.248,E1 17.7631,E2 529.8161} C_DIS
LIN {X 24.139,Y -128.9902,Z 158,A -78.9748,B 17.7335,C -0.286,E1 17.7694,E2 527.528} C_DIS
LIN {X 30.2509,Y -127.695,Z 158,A -77.0754,B 17.7339,C -0.2569,E1 17.7743,E2 525.7279} C_DIS
LIN {X 36.7455,Y -125.9788,Z 158,A -74.4209,B 17.734,C -0.2493,E1 17.7814,E2 523.1046} C_DIS
LIN {X 40.5285,Y -124.8146,Z 158,A -72.3687,B 17.7338,C -0.2634,E1 17.7869,E2 521.0117} C_DIS
LIN {X 44.0829,Y -123.6032,Z 158,A -70.8135,B 17.7338,C -0.2621,E1 17.791,E2 519.4652} C_DIS
LIN {X 47.0137,Y -122.5189,Z 158,A -69.4092,B 17.7338,C -0.2654,E1 17.7947,E2 518.0548} C_DIS
LIN {X 49.9276,Y -121.3612,Z 158,A -68.056,B 17.7338,C -0.2666,E1 17.7982,E2 516.7022} C_DIS
LIN {X 53.3815,Y -119.8803,Z 158,A -66.4625,B 17.7338,C -0.2671,E1 17.8023,E2 515.1127} C_DIS
LIN {X 56.3284,Y -118.5242,Z 158,A -64.4449,B 17.7334,C -0.2923,E1 17.8076,E2 513.0202} C_DIS
LIN {X 60.8123,Y -116.2872,Z 158,A -63.0558,B 17.7338,C -0.2649,E1 17.8108,E2 511.7263} C_DIS
LIN {X 63.8388,Y -114.6562,Z 158,A -61.3917,B 17.7337,C -0.2736,E1 17.8149,E2 510.0408} C_DIS
LIN {X 67.37,Y -112.6173,Z 158,A -59.1238,B 17.7333,C -0.2956,E1 17.8205,E2 507.7114} C_DIS
LIN {X 71.1155,Y -110.2908,Z 158,A -57.7257,B 17.7336,C -0.2786,E1 17.8236,E2 506.3754} C_DIS
LIN {X 74.3802,Y -108.1154,Z 158,A -55.9446,B 17.7336,C -0.2844,E1 17.8278,E2 504.5839} C_DIS
LIN {X 77.7745,Y -105.6999,Z 158,A -54.0575,B 17.7334,C -0.2906,E1 17.8321,E2 502.6862} C_DIS
LIN {X 83.2315,Y -101.4588,Z 158,A -51.1144,B 17.7334,C -0.2939,E1 17.8385,E2 499.7485} C_DIS
LIN {X 88.2201,Y -97.1522,Z 158,A -48.5782,B 17.7334,C -0.2868,E1 17.8438,E2 497.25} C_DIS
LIN {X 93.0071,Y -92.5798,Z 158,A -45.7668,B 17.7334,C -0.2902,E1 17.8494,E2 494.4447} C_DIS
LIN {X 97.1501,Y -88.2223,Z 158,A -43.0487,B 17.7333,C -0.2999,E1 17.8547,E2 491.7119} C_DIS
LIN {X 101.2422,Y -83.495,Z 158,A -40.0912,B 17.733,C -0.3155,E1 17.8601,E2 488.7232} C_DIS
LIN {X 103.0385,Y -81.2679,Z 158,A -38.2544,B 17.7325,C -0.3419,E1 17.8634,E2 486.8128} C_DIS
LIN {X 106.162,Y -77.1426,Z 158,A -36.4362,B 17.7327,C -0.3303,E1 17.8663,E2 485.0454} C_DIS
LIN {X 108.963,Y -73.1334,Z 158,A -34.5239,B 17.7327,C -0.3271,E1 17.8692,E2 483.1573} C_DIS
LIN {X 110.98,Y -70.0341,Z 158,A -32.8652,B 17.7327,C -0.3332,E1 17.8718,E2 481.4908} C_DIS
LIN {X 113.3386,Y -66.1501,Z 158,A -30.907,B 17.7327,C -0.3376,E1 17.8745,E2 479.5329} C_DIS
LIN {X 115.4348,Y -62.4201,Z 158,A -29.0197,B 17.7325,C -0.3435,E1 17.8771,E2 477.6406} C_DIS
LIN {X 117.3222,Y -58.7963,Z 158,A -27.3171,B 17.7325,C -0.3454,E1 17.8792,E2 475.9452} C_DIS
LIN {X 119.2104,Y -54.8613,Z 158,A -25.475,B 17.7325,C -0.3483,E1 17.8814,E2 474.1079} C_DIS
LIN {X 120.3643,Y -52.281,Z 158,A -23.6832,B 17.7319,C -0.3741,E1 17.8835,E2 472.2463} C_DIS
LIN {X 122.1411,Y -47.9818,Z 158,A -21.865,B 17.7319,C -0.3716,E1 17.8853,E2 470.4512} C_DIS
LIN {X 123.4479,Y -44.5135,Z 158,A -20.634,B 17.7322,C -0.3609,E1 17.8865,E2 469.2649} C_DIS
LIN {X 124.7703,Y -40.6673,Z 158,A -18.7691,B 17.732,C -0.3697,E1 17.8881,E2 467.3867} C_DIS
LIN {X 127.1707,Y -32.3804,Z 158,A -15.1483,B 17.7319,C -0.3752,E1 17.8909,E2 463.7781} C_DIS
LIN {X 127.825,Y -29.6967,Z 158,A -13.4315,B 17.7314,C -0.3993,E1 17.892,E2 461.9974} C_DIS
LIN {X 128.7603,Y -25.3416,Z 158,A -12.0759,B 17.7317,C -0.3816,E1 17.8927,E2 460.7107} C_DIS
LIN {X 129.7696,Y -19.5214,Z 158,A -9.3582,B 17.7315,C -0.3951,E1 17.894,E2 457.9726} C_DIS
LIN {X 130.273,Y -15.8094,Z 158,A -7.5057,B 17.7312,C -0.4088,E1 17.8946,E2 456.0912} C_DIS
LIN {X 130.6437,Y -12.3771,Z 158,A -6.3363,B 17.7313,C -0.4,E1 17.8949,E2 454.9607} C_DIS
LIN {X 130.9769,Y -8.1238,Z 158,A -4.469,B 17.7313,C -0.4059,E1 17.8953,E2 453.0902} C_DIS
LIN {X 131.1767,Y -3.6941,Z 158,A -2.5797,B 17.7311,C -0.41,E1 17.8955,E2 451.2038} C_DIS
LIN {X 131.2306,Y 0.1424,Z 158,A -0.7974,B 17.7309,C -0.4194,E1 17.8955,E2 449.4063} C_DIS
LIN {X 131.1591,Y 4.3269,Z 158,A 1.003,B 17.7309,C -0.424,E1 17.8954,E2 447.6066} C_DIS
LIN {X 130.9721,Y 8.2027,Z 158,A 2.5882,B 17.7308,C -0.4249,E1 17.8951,E2 446.0322} C_DIS
LIN {X 130.6404,Y 12.4111,Z 158,A 4.2851,B 17.7308,C -0.4247,E1 17.8947,E2 444.3504} C_DIS
LIN {X 130.3151,Y 15.4563,Z 158,A 5.7205,B 17.7306,C -0.4327,E1 17.8943,E2 442.9014} C_DIS
LIN {X 129.8876,Y 18.7119,Z 158,A 7.2809,B 17.7304,C -0.4421,E1 17.8937,E2 441.3238} C_DIS
LIN {X 129.1929,Y 23.0237,Z 158,A 9.6872,B 17.7297,C -0.4678,E1 17.8925,E2 438.8545} C_DIS
LIN {X 128.1914,Y 28.0713,Z 158,A 11.2177,B 17.7303,C -0.4459,E1 17.8916,E2 437.408} C_DIS
LIN {X 126.8784,Y 33.5088,Z 158,A 13.702,B 17.7301,C -0.4548,E1 17.89,E2 434.9156} C_DIS
LIN {X 126.097,Y 36.3417,Z 158,A 15.2813,B 17.7297,C -0.4703,E1 17.8887,E2 433.299} C_DIS
LIN {X 125.1199,Y 39.5729,Z 158,A 16.3518,B 17.73,C -0.4586,E1 17.8879,E2 432.2754} C_DIS
LIN {X 124.1141,Y 42.6225,Z 158,A 17.7557,B 17.7299,C -0.4627,E1 17.8866,E2 430.8697} C_DIS
LIN {X 122.9343,Y 45.9131,Z 158,A 19.1795,B 17.7299,C -0.4631,E1 17.8852,E2 429.4564} C_DIS
LIN {X 121.9558,Y 48.4566,Z 158,A 20.6153,B 17.7295,C -0.4761,E1 17.8837,E2 427.9898} C_DIS
LIN {X 120.4331,Y 52.122,Z 158,A 22.1912,B 17.7295,C -0.4747,E1 17.882,E2 426.4308} C_DIS
LIN {X 118.8739,Y 55.5889,Z 158,A 23.8585,B 17.7295,C -0.4796,E1 17.8801,E2 424.7609} C_DIS
LIN {X 117.1526,Y 59.1295,Z 158,A 25.6386,B 17.7293,C -0.4866,E1 17.8779,E2 422.9716} C_DIS
LIN {X 115.3758,Y 62.529,Z 158,A 27.3337,B 17.7291,C -0.4919,E1 17.8757,E2 421.2725} C_DIS
LIN {X 113.3109,Y 66.1971,Z 158,A 29.1518,B 17.7291,C -0.4959,E1 17.8731,E2 419.455} C_DIS
LIN {X 111.0326,Y 69.9507,Z 158,A 31.0197,B 17.7289,C -0.4989,E1 17.8704,E2 417.5911} C_DIS
LIN {X 108.7338,Y 73.4732,Z 158,A 32.8211,B 17.7289,C -0.5021,E1 17.8676,E2 415.7923} C_DIS
LIN {X 106.3233,Y 76.9201,Z 158,A 34.7099,B 17.7287,C -0.5086,E1 17.8645,E2 413.8957} C_DIS
LIN {X 103.5171,Y 80.6576,Z 158,A 36.7403,B 17.7285,C -0.513,E1 17.8611,E2 411.8649} C_DIS
LIN {X 100.7825,Y 84.0491,Z 158,A 38.6305,B 17.7285,C -0.5169,E1 17.8577,E2 409.9746} C_DIS
LIN {X 98.1932,Y 87.06,Z 158,A 40.5481,B 17.7281,C -0.5279,E1 17.8542,E2 408.0338} C_DIS
LIN {X 95.9859,Y 89.4875,Z 158,A 41.8034,B 17.7282,C -0.5242,E1 17.8518,E2 406.7987} C_DIS
LIN {X 92.7322,Y 92.8557,Z 158,A 43.8076,B 17.7282,C -0.5269,E1 17.8479,E2 404.798} C_DIS
LIN {X 89.5382,Y 95.9388,Z 158,A 45.6963,B 17.7281,C -0.529,E1 17.8441,E2 402.914} C_DIS
LIN {X 86.2691,Y 98.8886,Z 158,A 47.614,B 17.728,C -0.5325,E1 17.8401,E2 400.9959} C_DIS
LIN {X 83.9639,Y 100.8539,Z 158,A 49.2674,B 17.7275,C -0.5477,E1 17.8364,E2 399.3022} C_DIS
LIN {X 80.9917,Y 103.2552,Z 158,A 50.6836,B 17.7277,C -0.541,E1 17.8334,E2 397.9154} C_DIS
LIN {X 77.3513,Y 106.0108,Z 158,A 52.6193,B 17.7277,C -0.5423,E1 17.8291,E2 395.9856} C_DIS
LIN {X 73.6938,Y 108.5845,Z 158,A 54.5289,B 17.7277,C -0.5439,E1 17.8247,E2 394.0804} C_DIS
LIN {X 69.9359,Y 111.042,Z 158,A 56.477,B 17.7276,C -0.5465,E1 17.8201,E2 392.1331} C_DIS
LIN {X 66.3155,Y 113.2414,Z 158,A 58.3301,B 17.7275,C -0.5493,E1 17.8157,E2 390.2791} C_DIS
LIN {X 62.6498,Y 115.31,Z 158,A 60.1682,B 17.7275,C -0.5519,E1 17.8112,E2 388.4404} C_DIS
LIN {X 59.4167,Y 117.0064,Z 158,A 61.6711,B 17.7275,C -0.5505,E1 17.8075,E2 386.9479} C_DIS
LIN {X 55.5895,Y 118.8737,Z 158,A 63.5711,B 17.7273,C -0.5543,E1 17.8027,E2 385.0429} C_DIS
LIN {X 52.2873,Y 120.3616,Z 158,A 65.1378,B 17.7273,C -0.5555,E1 17.7987,E2 383.4776} C_DIS
LIN {X 48.9313,Y 121.7645,Z 158,A 66.6192,B 17.7273,C -0.5532,E1 17.7949,E2 382.0088} C_DIS
LIN {X 45.9526,Y 122.9195,Z 158,A 68.0719,B 17.7273,C -0.5568,E1 17.7911,E2 380.5492} C_DIS
LIN {X 42.2285,Y 124.2507,Z 158,A 69.9078,B 17.7271,C -0.5623,E1 17.7862,E2 378.7005} C_DIS
LIN {X 38.5336,Y 125.4434,Z 158,A 71.218,B 17.7275,C -0.5495,E1 17.7828,E2 377.4357} C_DIS
LIN {X 34.1725,Y 126.7014,Z 158,A 73.4788,B 17.7271,C -0.5612,E1 17.7767,E2 375.1422} C_DIS
LIN {X 31.0612,Y 127.4997,Z 158,A 74.8535,B 17.7271,C -0.561,E1 17.7729,E2 373.771} C_DIS
LIN {X 26.4804,Y 128.5293,Z 158,A 77.0947,B 17.7269,C -0.5691,E1 17.7668,E2 371.5076} C_DIS
LIN {X 21.7451,Y 129.4144,Z 158,A 78.9941,B 17.7271,C -0.5626,E1 17.7616,E2 369.6328} C_DIS
LIN {X 17.0757,Y 130.1128,Z 158,A 81.1385,B 17.727,C -0.5662,E1 17.7556,E2 367.4792} C_DIS
LIN {X 13.1593,Y 130.5686,Z 158,A 82.8651,B 17.727,C -0.5667,E1 17.7509,E2 365.7526} C_DIS
LIN {X 8.8737,Y 130.93,Z 158,A 84.7877,B 17.7269,C -0.5686,E1 17.7455,E2 363.8254} C_DIS
LIN {X 4.8854,Y 131.1379,Z 158,A 86.4812,B 17.7269,C -0.5668,E1 17.7408,E2 362.1385} C_DIS
LIN {X 0.4702,Y 131.2281,Z 158,A 88.369,B 17.7269,C -0.5652,E1 17.7355,E2 360.2563} C_DIS
LIN {X -3.3268,Y 131.1869,Z 158,A 90.0114,B 17.727,C -0.5643,E1 17.7309,E2 358.6166} C_DIS
LIN {X -6.9978,Y 131.0426,Z 158,A 91.5774,B 17.727,C -0.5625,E1 17.7266,E2 357.056} C_DIS
LIN {X -11.0478,Y 130.7627,Z 158,A 93.4099,B 17.727,C -0.564,E1 17.7215,E2 355.2175} C_DIS
LIN {X -15.2613,Y 130.3382,Z 158,A 95.3755,B 17.727,C -0.5673,E1 17.716,E2 353.2393} C_DIS
LIN {X -20.7086,Y 129.5858,Z 158,A 98.5693,B 17.7261,C -0.5942,E1 17.7069,E2 349.9532} C_DIS
LIN {X -27.1745,Y 128.385,Z 158,A 100.3647,B 17.7273,C -0.5539,E1 17.7024,E2 348.2874} C_DIS
LIN {X -33.1458,Y 126.9752,Z 158,A 103.2516,B 17.7272,C -0.5589,E1 17.6945,E2 345.3783} C_DIS
LIN {X -36.7243,Y 125.985,Z 158,A 104.5843,B 17.7275,C -0.5473,E1 17.691,E2 344.0808} C_DIS
LIN {X -40.3543,Y 124.8703,Z 158,A 106.4863,B 17.7273,C -0.554,E1 17.6858,E2 342.1517} C_DIS
LIN {X -44.0273,Y 123.6232,Z 158,A 108.1829,B 17.7273,C -0.5522,E1 17.6814,E2 340.4562} C_DIS
LIN {X -47.0103,Y 122.5202,Z 158,A 109.6605,B 17.7273,C -0.5536,E1 17.6775,E2 338.9695} C_DIS
LIN {X -54.4725,Y 119.3902,Z 158,A 113.2034,B 17.7275,C -0.5492,E1 17.6684,E2 335.4291} C_DIS
LIN {X -57.8538,Y 117.7871,Z 158,A 114.5502,B 17.7278,C -0.537,E1 17.6651,E2 334.1176} C_DIS
LIN {X -62.3651,Y 115.4643,Z 158,A 117.0891,B 17.7276,C -0.5446,E1 17.6587,E2 331.5433} C_DIS
LIN {X -66.2812,Y 113.2616,Z 158,A 119.0214,B 17.7277,C -0.5404,E1 17.6541,E2 329.6167} C_DIS
LIN {X -69.8946,Y 111.068,Z 158,A 120.8878,B 17.7278,C -0.5379,E1 17.6496,E2 327.7499} C_DIS
LIN {X -73.6112,Y 108.6403,Z 158,A 122.8305,B 17.7279,C -0.5346,E1 17.6451,E2 325.809} C_DIS
LIN {X -77.325,Y 106.0298,Z 158,A 124.8612,B 17.7279,C -0.5325,E1 17.6405,E2 323.775} C_DIS
LIN {X -80.7899,Y 103.4139,Z 158,A 126.7755,B 17.7281,C -0.5294,E1 17.6363,E2 321.8608} C_DIS
LIN {X -84.3623,Y 100.5203,Z 158,A 128.7172,B 17.7282,C -0.523,E1 17.6321,E2 319.9293} C_DIS
LIN {X -87.4047,Y 97.8866,Z 158,A 130.4559,B 17.7284,C -0.5186,E1 17.6285,E2 318.195} C_DIS
LIN {X -91.5315,Y 94.0396,Z 158,A 132.9954,B 17.7284,C -0.5158,E1 17.6233,E2 315.6498} C_DIS
LIN {X -94.5899,Y 90.9628,Z 158,A 134.9081,B 17.7286,C -0.512,E1 17.6196,E2 313.7375} C_DIS
LIN {X -97.4741,Y 87.8653,Z 158,A 136.7861,B 17.7286,C -0.5087,E1 17.616,E2 311.8584} C_DIS
LIN {X -100.3125,Y 84.61,Z 158,A 138.6966,B 17.7288,C -0.5049,E1 17.6126,E2 309.9476} C_DIS
LIN {X -102.9871,Y 81.3333,Z 158,A 140.5752,B 17.7288,C -0.5014,E1 17.6093,E2 308.0679} C_DIS
LIN {X -105.7662,Y 77.6842,Z 158,A 142.514,B 17.729,C -0.4942,E1 17.606,E2 306.1394} C_DIS
LIN {X -108.1663,Y 74.306,Z 158,A 144.3037,B 17.7292,C -0.4888,E1 17.6032,E2 304.3545} C_DIS
LIN {X -110.3157,Y 71.0769,Z 158,A 146.0826,B 17.7292,C -0.4872,E1 17.6005,E2 302.5681} C_DIS
LIN {X -112.4885,Y 67.5856,Z 158,A 147.9004,B 17.7293,C -0.4831,E1 17.5978,E2 300.7502} C_DIS
LIN {X -114.4123,Y 64.2741,Z 158,A 150.1256,B 17.729,C -0.4969,E1 17.5947,E2 298.4622} C_DIS
LIN {X -116.7313,Y 59.957,Z 158,A 151.4927,B 17.7298,C -0.4652,E1 17.593,E2 297.1892} C_DIS
LIN {X -118.3523,Y 56.6883,Z 158,A 152.9645,B 17.73,C -0.4568,E1 17.5913,E2 295.734} C_DIS
LIN {X -119.5472,Y 54.1263,Z 158,A 154.4839,B 17.7299,C -0.4626,E1 17.5894,E2 294.183} C_DIS
LIN {X -120.9204,Y 50.9832,Z 158,A 156.0124,B 17.7299,C -0.4593,E1 17.5877,E2 292.6531} C_DIS
LIN {X -122.4397,Y 47.2173,Z 158,A 157.8169,B 17.7301,C -0.4552,E1 17.5859,E2 290.8475} C_DIS
LIN {X -123.9008,Y 43.2378,Z 158,A 159.7396,B 17.7301,C -0.4521,E1 17.5841,E2 288.9191} C_DIS
LIN {X -125.216,Y 39.2721,Z 158,A 161.635,B 17.7302,C -0.449,E1 17.5825,E2 287.0182} C_DIS
LIN {X -126.3021,Y 35.6191,Z 158,A 163.2003,B 17.7304,C -0.4408,E1 17.5813,E2 285.4667} C_DIS
LIN {X -127.1086,Y 32.6253,Z 158,A 164.627,B 17.7304,C -0.4391,E1 17.5802,E2 284.0335} C_DIS
LIN {X -128.3733,Y 27.2287,Z 158,A 166.9716,B 17.7307,C -0.4292,E1 17.5788,E2 281.7014} C_DIS
LIN {X -128.8982,Y 24.62,Z 158,A 168.5304,B 17.7305,C -0.4388,E1 17.578,E2 280.0975} C_DIS
LIN {X -129.5432,Y 20.973,Z 158,A 169.8975,B 17.7308,C -0.4256,E1 17.5774,E2 278.7622} C_DIS
LIN {X -130.1531,Y 16.7684,Z 158,A 171.6687,B 17.731,C -0.4171,E1 17.5767,E2 277.0035} C_DIS
LIN {X -130.5793,Y 13.0476,Z 158,A 173.3154,B 17.731,C -0.4125,E1 17.5762,E2 275.3579} C_DIS
LIN {X -131.0058,Y 7.6548,Z 158,A 175.7072,B 17.7312,C -0.4061,E1 17.5757,E2 272.966} C_DIS
LIN {X -131.2308,Y -0.1101,Z 158,A 179.8629,B 17.7309,C -0.421,E1 17.5756,E2 268.7246} C_DIS
LIN {X -131.1135,Y -5.5116,Z 158,A -178.4763,B 17.7316,C -0.3906,E1 17.5757,E2 267.1499} C_DIS
LIN {X -130.7073,Y -11.7041,Z 158,A -175.5534,B 17.7316,C -0.3893,E1 17.5763,E2 264.2055} C_DIS
LIN {X -129.7729,Y -19.4999,Z 158,A -172.2333,B 17.7319,C -0.3753,E1 17.5775,E2 260.9028} C_DIS
LIN {X -129.0087,Y -24.042,Z 158,A -169.6577,B 17.7316,C -0.388,E1 17.5788,E2 258.2628} C_DIS
LIN {X -128.0383,Y -28.7627,Z 158,A -168.0942,B 17.7321,C -0.3637,E1 17.5797,E2 256.7663} C_DIS
LIN {X -127.2149,Y -32.2062,Z 158,A -166.5859,B 17.7322,C -0.3579,E1 17.5807,E2 255.2643} C_DIS
LIN {X -126.3333,Y -35.5075,Z 158,A -165.0773,B 17.7322,C -0.3541,E1 17.5818,E2 253.7555} C_DIS
LIN {X -125.1314,Y -39.5368,Z 158,A -163.2176,B 17.7324,C -0.3496,E1 17.5834,E2 251.8951} C_DIS
LIN {X -124.035,Y -42.8507,Z 158,A -161.7517,B 17.7324,C -0.3433,E1 17.5847,E2 250.438} C_DIS
LIN {X -121.3597,Y -49.9314,Z 158,A -158.2582,B 17.7326,C -0.3402,E1 17.5882,E2 246.926} C_DIS
LIN {X -117.5614,Y -58.3113,Z 158,A -154.2882,B 17.7328,C -0.3276,E1 17.5929,E2 242.966} C_DIS
LIN {X -115.5525,Y -62.201,Z 158,A -152.3674,B 17.7328,C -0.3228,E1 17.5953,E2 241.0462} C_DIS
LIN {X -111.917,Y -68.5269,Z 158,A -149.4725,B 17.7332,C -0.3048,E1 17.5994,E2 238.1889} C_DIS
LIN {X -108.1182,Y -74.3761,Z 158,A -146.0617,B 17.7332,C -0.3094,E1 17.6047,E2 234.7376} C_DIS
LIN {X -105.6497,Y -77.8428,Z 158,A -144.1631,B 17.7332,C -0.3063,E1 17.6077,E2 232.8359} C_DIS
LIN {X -103.5933,Y -80.5593,Z 158,A -142.2601,B 17.733,C -0.317,E1 17.6111,E2 230.8843} C_DIS
LIN {X -100.9857,Y -83.8048,Z 158,A -140.8977,B 17.7333,C -0.2973,E1 17.6134,E2 229.5779} C_DIS
LIN {X -96.7325,Y -88.6802,Z 158,A -137.9702,B 17.7333,C -0.2946,E1 17.6189,E2 226.6403} C_DIS
LIN {X -93.6045,Y -91.9758,Z 158,A -136.0516,B 17.7334,C -0.2882,E1 17.6226,E2 224.7308} C_DIS
LIN {X -87.5959,Y -97.7154,Z 158,A -132.7358,B 17.7337,C -0.2701,E1 17.6292,E2 221.4545} C_DIS
LIN {X -81.685,Y -102.7078,Z 158,A -128.924,B 17.7336,C -0.2787,E1 17.6375,E2 217.593} C_DIS
LIN {X -78.1651,Y -105.4116,Z 158,A -126.9837,B 17.7336,C -0.2755,E1 17.6418,E2 215.6534} C_DIS
LIN {X -74.6892,Y -107.9026,Z 158,A -125.1035,B 17.7336,C -0.2729,E1 17.6461,E2 213.7724} C_DIS
LIN {X -71.1643,Y -110.2592,Z 158,A -123.4536,B 17.7338,C -0.263,E1 17.6499,E2 212.1473} C_DIS
LIN {X -68.1748,Y -112.1314,Z 158,A -121.784,B 17.7338,C -0.2652,E1 17.6539,E2 210.4627} C_DIS
LIN {X -64.7916,Y -114.1204,Z 158,A -119.9902,B 17.7338,C -0.2657,E1 17.6582,E2 208.6597} C_DIS
LIN {X -61.2139,Y -116.0764,Z 158,A -118.3793,B 17.7339,C -0.2574,E1 17.6621,E2 207.0695} C_DIS
LIN {X -58.241,Y -117.5961,Z 158,A -116.7459,B 17.7339,C -0.2618,E1 17.6663,E2 205.4152} C_DIS
LIN {X -54.9535,Y -119.1678,Z 158,A -115.1722,B 17.7339,C -0.2593,E1 17.6702,E2 203.8439} C_DIS
LIN {X -50.9315,Y -120.942,Z 158,A -113.3645,B 17.7339,C -0.2533,E1 17.6748,E2 202.0499} C_DIS
LIN {X -47.6758,Y -122.2615,Z 158,A -111.7079,B 17.7339,C -0.2562,E1 17.6792,E2 200.3785} C_DIS
LIN {X -43.753,Y -123.7221,Z 158,A -109.8326,B 17.7339,C -0.2562,E1 17.6841,E2 198.4976} C_DIS
LIN {X -40.6226,Y -124.7845,Z 158,A -108.0011,B 17.7337,C -0.269,E1 17.6891,E2 196.6191} C_DIS
LIN {X -36.7363,Y -125.9814,Z 158,A -106.6756,B 17.734,C -0.2516,E1 17.6925,E2 195.3478} C_DIS
LIN {X -32.7606,Y -127.0742,Z 158,A -104.7978,B 17.734,C -0.2532,E1 17.6976,E2 193.4606} C_DIS
LIN {X -29.2737,Y -127.9216,Z 158,A -103.2451,B 17.734,C -0.2519,E1 17.7018,E2 191.9093} C_DIS
LIN {X -24.8351,Y -128.8571,Z 158,A -101.3429,B 17.734,C -0.2482,E1 17.707,E2 190.0161} C_DIS
LIN {X -21.8912,Y -129.39,Z 158,A -99.8933,B 17.734,C -0.2529,E1 17.711,E2 188.5489} C_DIS
LIN {X -17.1451,Y -130.1037,Z 158,A -97.9098,B 17.734,C -0.2483,E1 17.7165,E2 186.5782} C_DIS
LIN {X -12.853,Y -130.598,Z 158,A -96.0468,B 17.734,C -0.2472,E1 17.7217,E2 184.7175} C_DIS
LIN {X -9.3016,Y -130.8988,Z 158,A -94.4345,B 17.734,C -0.2491,E1 17.7262,E2 183.0978} C_DIS
LIN {X -4.9327,Y -131.136,Z 158,A -92.5245,B 17.734,C -0.2491,E1 17.7315,E2 181.187} C_DIS
LIN {X -1.3111,Y -131.2235,Z 158,A -91.0373,B 17.734,C -0.2459,E1 17.7356,E2 179.7105} C_DIS
LIN {X 0.9148,Y -131.2224,Z 158,A -90.2085,B 17.7341,C -0.2408,E1 17.7379,E2 178.8984} C_DIS
Enddeposition()
LIN {X 0.9148,Y -131.2224,Z 158,A -90.2085,B 17.7341,C -0.2408,E1 17.7379,E2 178.8984} C_DIS
Startdeposition()
$VEL.CP = VEL_PRINT
LIN {X -1.1529,Y -130.295,Z 158,A -90.8408,B 14.7772,C 0.0463,E1 14.7751,E2 180.3966} C_DIS
LIN {X -5.895,Y -130.1675,Z 158,A -92.7202,B 14.7772,C 0.0402,E1 14.77,E2 182.2527} C_DIS
LIN {X -8.1847,Y -130.0421,Z 158,A -93.8834,B 14.7772,C 0.0448,E1 14.7667,E2 183.4345} C_DIS
LIN {X -12.4769,Y -129.7005,Z 158,A -95.73,B 14.7772,C 0.0432,E1 14.7615,E2 185.2763} C_DIS
LIN {X -16.1546,Y -129.2959,Z 158,A -97.2909,B 14.7772,C 0.041,E1 14.7572,E2 186.8299} C_DIS
LIN {X -18.954,Y -128.9143,Z 158,A -98.8021,B 14.7772,C 0.0486,E1 14.753,E2 188.3732} C_DIS
LIN {X -23.1999,Y -128.2173,Z 158,A -100.5016,B 14.7772,C 0.0422,E1 14.7484,E2 190.0505} C_DIS
LIN {X -28.2339,Y -127.2056,Z 158,A -102.6927,B 14.7772,C 0.0392,E1 14.7424,E2 192.2344} C_DIS
LIN {X -32.1731,Y -126.2645,Z 158,A -104.5461,B 14.7772,C 0.0403,E1 14.7373,E2 194.0965} C_DIS
LIN {X -35.7535,Y -125.2996,Z 158,A -106.1276,B 14.7772,C 0.0378,E1 14.7331,E2 195.6725} C_DIS
LIN {X -39.8481,Y -124.0564,Z 158,A -108.0761,B 14.7772,C 0.0383,E1 14.7279,E2 197.629} C_DIS
LIN {X -44.3899,Y -122.5046,Z 158,A -110.0949,B 14.7772,C 0.0339,E1 14.7226,E2 199.6372} C_DIS
LIN {X -48.0009,Y -121.1375,Z 158,A -111.824,B 14.7772,C 0.0332,E1 14.7181,E2 201.3701} C_DIS
LIN {X -51.0115,Y -119.9008,Z 158,A -113.4952,B 14.7772,C 0.0386,E1 14.7137,E2 203.0694} C_DIS
LIN {X -54.9402,Y -118.15,Z 158,A -115.1983,B 14.7772,C 0.0311,E1 14.7094,E2 204.7503} C_DIS
LIN {X -58.4977,Y -116.4314,Z 158,A -116.9362,B 14.7772,C 0.0291,E1 14.7051,E2 206.4881} C_DIS
LIN {X -61.9634,Y -114.6252,Z 158,A -118.6556,B 14.7772,C 0.0269,E1 14.7008,E2 208.2074} C_DIS
LIN {X -65.4253,Y -112.6847,Z 158,A -120.3369,B 14.7772,C 0.0227,E1 14.6968,E2 209.8808} C_DIS
LIN {X -70.5422,Y -109.5544,Z 158,A -122.9753,B 14.7772,C 0.0189,E1 14.6905,E2 212.5188} C_DIS
LIN {X -73.4565,Y -107.6222,Z 158,A -124.491,B 14.7772,C 0.0159,E1 14.687,E2 214.0315} C_DIS
LIN {X -75.4573,Y -106.2292,Z 158,A -125.6974,B 14.7772,C 0.018,E1 14.6842,E2 215.2533} C_DIS
LIN {X -78.7615,Y -103.8028,Z 158,A -127.5325,B 14.7772,C 0.0159,E1 14.6801,E2 217.0916} C_DIS
LIN {X -83.5642,Y -99.9768,Z 158,A -130.2185,B 14.7772,C 0.0107,E1 14.6742,E2 219.775} C_DIS
LIN {X -86.3227,Y -97.6047,Z 158,A -131.8849,B 14.7772,C 0.0096,E1 14.6707,E2 221.4485} C_DIS
LIN {X -89.2467,Y -94.9387,Z 158,A -133.9778,B 14.7772,C 0.0159,E1 14.6664,E2 223.5816} C_DIS
LIN {X -91.8856,Y -92.3868,Z 158,A -135.2781,B 14.7772,C 0.004,E1 14.6638,E2 224.8445} C_DIS
LIN {X -94.8756,Y -89.3136,Z 158,A -137.3302,B 14.7772,C 0.0047,E1 14.6598,E2 226.915} C_DIS
LIN {X -98.277,Y -85.5566,Z 158,A -139.3965,B 14.7772,C -0.0045,E1 14.6561,E2 228.9611} C_DIS
LIN {X -101.0474,Y -82.2664,Z 158,A -141.4043,B 14.7772,C -0.0056,E1 14.6525,E2 230.9813} C_DIS
LIN {X -103.3317,Y -79.3784,Z 158,A -142.9514,B 14.7772,C -0.0112,E1 14.6498,E2 232.519} C_DIS
LIN {X -105.5247,Y -76.4384,Z 158,A -144.5956,B 14.7772,C -0.0142,E1 14.6471,E2 234.1657} C_DIS
LIN {X -108.969,Y -71.4431,Z 158,A -147.3169,B 14.7772,C -0.0192,E1 14.6428,E2 236.8912} C_DIS
LIN {X -111.2575,Y -67.8247,Z 158,A -149.1794,B 14.7772,C -0.0244,E1 14.6401,E2 238.7499} C_DIS
LIN {X -113.6074,Y -63.8095,Z 158,A -151.0236,B 14.7772,C -0.035,E1 14.6375,E2 240.569} C_DIS
LIN {X -114.8209,Y -61.5991,Z 158,A -152.3176,B 14.7772,C -0.0329,E1 14.6358,E2 241.8836} C_DIS
LIN {X -116.5316,Y -58.2983,Z 158,A -154.3462,B 14.7772,C -0.0266,E1 14.6332,E2 243.9563} C_DIS
LIN {X -118.1064,Y -55.0346,Z 158,A -155.3651,B 14.7772,C -0.0462,E1 14.6321,E2 244.9073} C_DIS
LIN {X -119.1598,Y -52.7163,Z 158,A -156.6798,B 14.7772,C -0.044,E1 14.6305,E2 246.2436} C_DIS
LIN {X -120.6084,Y -49.3135,Z 158,A -158.4849,B 14.7772,C -0.0437,E1 14.6286,E2 248.0678} C_DIS
LIN {X -122.6231,Y -44.0612,Z 158,A -160.7212,B 14.7772,C -0.0569,E1 14.6264,E2 250.2743} C_DIS
LIN {X -123.6735,Y -41.0206,Z 158,A -162.2122,B 14.7772,C -0.0588,E1 14.625,E2 251.7728} C_DIS
LIN {X -124.6544,Y -37.9359,Z 158,A -163.6723,B 14.7772,C -0.0618,E1 14.6238,E2 253.2357} C_DIS
LIN {X -125.6845,Y -34.3771,Z 158,A -165.4159,B 14.7772,C -0.0634,E1 14.6225,E2 254.9908} C_DIS
LIN {X -126.6689,Y -30.5422,Z 158,A -167.1027,B 14.7772,C -0.0699,E1 14.6214,E2 256.6694} C_DIS
LIN {X -127.6496,Y -26.1431,Z 158,A -168.9096,B 14.7771,C -0.0803,E1 14.6203,E2 258.4539} C_DIS
LIN {X -128.2752,Y -22.8765,Z 158,A -170.6448,B 14.7771,C -0.0774,E1 14.6194,E2 260.219} C_DIS
LIN {X -128.952,Y -18.69,Z 158,A -172.681,B 14.7771,C -0.0784,E1 14.6185,E2 262.2728} C_DIS
LIN {X -129.4365,Y -14.9758,Z 158,A -174.1006,B 14.7771,C -0.0893,E1 14.6181,E2 263.6644} C_DIS
LIN {X -130.025,Y -8.4628,Z 158,A -177.0939,B 14.7771,C -0.0947,E1 14.6174,E2 266.6679} C_DIS
LIN {X -130.2222,Y -4.5184,Z 158,A -179.479,B 14.7771,C -0.083,E1 14.6171,E2 269.1251} C_DIS
LIN {X -130.2984,Y 0.6417,Z 158,A 178.4465,B 14.7771,C -0.0949,E1 14.6171,E2 271.1746} C_DIS
LIN {X -130.2143,Y 4.7201,Z 158,A 177.3063,B 14.7768,C -0.1174,E1 14.6172,E2 272.2378} C_DIS
LIN {X -129.9386,Y 9.69,Z 158,A 174.9368,B 14.7768,C -0.1193,E1 14.6176,E2 274.6254} C_DIS
LIN {X -129.6198,Y 13.304,Z 158,A 173.3687,B 14.7768,C -0.1248,E1 14.618,E2 276.1884} C_DIS
LIN {X -129.2317,Y 16.6472,Z 158,A 171.8729,B 14.7768,C -0.1288,E1 14.6185,E2 277.6841} C_DIS
LIN {X -128.7452,Y 20.064,Z 158,A 170.1791,B 14.7768,C -0.1287,E1 14.6192,E2 279.3962} C_DIS
LIN {X -128.0428,Y 24.1454,Z 158,A 168.5548,B 14.7767,C -0.1393,E1 14.62,E2 280.9955} C_DIS
LIN {X -127.5609,Y 26.579,Z 158,A 167.3592,B 14.7767,C -0.1398,E1 14.6207,E2 282.2019} C_DIS
LIN {X -127.0035,Y 29.1197,Z 158,A 166.0748,B 14.7767,C -0.1395,E1 14.6215,E2 283.5009} C_DIS
LIN {X -126.066,Y 32.9487,Z 158,A 164.4868,B 14.7766,C -0.1484,E1 14.6225,E2 285.07} C_DIS
LIN {X -125.3807,Y 35.4633,Z 158,A 163.3045,B 14.7766,C -0.1508,E1 14.6234,E2 286.2549} C_DIS
LIN {X -124.3817,Y 38.8266,Z 158,A 161.7124,B 14.7766,C -0.154,E1 14.6247,E2 287.8508} C_DIS
LIN {X -123.5679,Y 41.3379,Z 158,A 160.5209,B 14.7765,C -0.1565,E1 14.6258,E2 289.0441} C_DIS
LIN {X -122.4935,Y 44.4208,Z 158,A 159.0517,B 14.7765,C -0.1598,E1 14.6271,E2 290.5153} C_DIS
LIN {X -120.9817,Y 48.3874,Z 158,A 157.3444,B 14.7764,C -0.1693,E1 14.6288,E2 292.202} C_DIS
LIN {X -120.0493,Y 50.6576,Z 158,A 156.146,B 14.7764,C -0.1692,E1 14.6301,E2 293.4126} C_DIS
LIN {X -118.6417,Y 53.8746,Z 158,A 154.5478,B 14.7764,C -0.172,E1 14.632,E2 295.015} C_DIS
LIN {X -117.5034,Y 56.3095,Z 158,A 153.4378,B 14.7763,C -0.1772,E1 14.6333,E2 296.1153} C_DIS
LIN {X -116.3209,Y 58.7146,Z 158,A 151.738,B 14.7763,C -0.1667,E1 14.6355,E2 297.873} C_DIS
LIN {X -114.5413,Y 62.1175,Z 158,A 150.331,B 14.7763,C -0.1786,E1 14.6373,E2 299.2458} C_DIS
LIN {X -112.7082,Y 65.3847,Z 158,A 148.6707,B 14.7762,C -0.1827,E1 14.6396,E2 300.9055} C_DIS
LIN {X -110.796,Y 68.5758,Z 158,A 147.0283,B 14.7762,C -0.1868,E1 14.642,E2 302.5466} C_DIS
LIN {X -108.5527,Y 72.0743,Z 158,A 145.209,B 14.7761,C -0.1917,E1 14.6447,E2 304.3626} C_DIS
LIN {X -106.1884,Y 75.5144,Z 158,A 143.3185,B 14.7761,C -0.1949,E1 14.6478,E2 306.257} C_DIS
LIN {X -103.4852,Y 79.1776,Z 158,A 141.4631,B 14.7759,C -0.2038,E1 14.6509,E2 308.0932} C_DIS
LIN {X -101.2528,Y 82.0136,Z 158,A 139.7135,B 14.7759,C -0.2032,E1 14.6539,E2 309.8594} C_DIS
LIN {X -98.452,Y 85.3559,Z 158,A 137.7767,B 14.7759,C -0.2072,E1 14.6574,E2 311.796} C_DIS
LIN {X -95.5648,Y 88.5761,Z 158,A 135.8785,B 14.7759,C -0.2117,E1 14.661,E2 313.6915} C_DIS
LIN {X -92.6931,Y 91.5774,Z 158,A 133.9819,B 14.7758,C -0.2139,E1 14.6647,E2 315.5939} C_DIS
LIN {X -89.2494,Y 94.9362,Z 158,A 132.0734,B 14.7756,C -0.224,E1 14.6685,E2 317.4763} C_DIS
LIN {X -87.0198,Y 96.9838,Z 158,A 130.5745,B 14.7756,C -0.2223,E1 14.6716,E2 318.9927} C_DIS
LIN {X -83.9662,Y 99.6395,Z 158,A 128.7648,B 14.7756,C -0.225,E1 14.6755,E2 320.8039} C_DIS
LIN {X -80.7187,Y 102.2881,Z 158,A 126.8924,B 14.7756,C -0.2278,E1 14.6796,E2 322.6775} C_DIS
LIN {X -77.4547,Y 104.7817,Z 158,A 125.1861,B 14.7755,C -0.234,E1 14.6833,E2 324.3705} C_DIS
LIN {X -74.1741,Y 107.1288,Z 158,A 123.4425,B 14.7755,C -0.238,E1 14.6873,E2 326.1087} C_DIS
LIN {X -71.5357,Y 108.908,Z 158,A 121.8885,B 14.7755,C -0.2362,E1 14.6909,E2 327.6788} C_DIS
LIN {X -68.435,Y 110.8831,Z 158,A 120.2619,B 14.7755,C -0.2386,E1 14.6948,E2 329.3049} C_DIS
LIN {X -64.7442,Y 113.0775,Z 158,A 118.127,B 14.7755,C -0.2349,E1 14.7,E2 331.466} C_DIS
LIN {X -61.784,Y 114.7216,Z 158,A 116.9517,B 14.7753,C -0.2458,E1 14.7028,E2 332.6041} C_DIS
LIN {X -58.4977,Y 116.4314,Z 158,A 115.373,B 14.7753,C -0.2495,E1 14.7067,E2 334.1754} C_DIS
LIN {X -56.0497,Y 117.6275,Z 158,A 114.0283,B 14.7753,C -0.2472,E1 14.7101,E2 335.5357} C_DIS
LIN {X -52.0543,Y 119.4499,Z 158,A 111.9244,B 14.7753,C -0.2449,E1 14.7155,E2 337.6575} C_DIS
LIN {X -48.288,Y 121.0218,Z 158,A 110.3874,B 14.7752,C -0.2542,E1 14.7194,E2 339.1635} C_DIS
LIN {X -45.3675,Y 122.1463,Z 158,A 108.9849,B 14.7752,C -0.2551,E1 14.7231,E2 340.5679} C_DIS
Enddeposition()
END
